  	 11:CASE GVL.mb_Output_Registers[GVL.WATERHARDWARETYPE] OF
		GVL.SWPWTR_TIME:
			//GVL.mb_Output_Registers[GVL.REALTIME_PLC_A2D] :=	0;	//nothing to read with FB circuit, just move motor
			IF GVL.mb_Output_Coils[GVL.REALTIME_ADVANCE] THEN		//move the motor forward
				IF TRUE THEN							//test the FB for limit - can't do this, pass through
					GVL_IO.WaterMotorFwd[FTN1] := TRUE;				// turn on the advance output
					GVL_IO.WaterMotorRvs[FTN1] := FALSE;
					wCycleCount := wCycleCount + 1;
					IF wCycleCount > wMotorTimeOn THEN				//done with timer?
						GVL_IO.WaterMotorFwd[FTN1] := FALSE;		//turn off outputs
						GVL_IO.WaterMotorRvs[FTN1] := FALSE;
						GVL.mb_Output_Coils[GVL.REALTIME_ADVANCE] := FALSE; // reset the advance boolean
						wCycleCount := 0;					//reset the timer counter						
					END_IF
				END_IF
			END_IF
			IF GVL.mb_Output_Coils[GVL.REALTIME_RETARD] THEN
				IF TRUE THEN							//test the FB for limit - can't do this, pass through
					GVL_IO.WaterMotorFwd[FTN1] := FALSE;				// turn on the reverse output
					GVL_IO.WaterMotorRvs[FTN1] := TRUE;
					wCycleCount := wCycleCount + 1;
					IF wCycleCount > wMotorTimeOn THEN				//done with timer?
						GVL_IO.WaterMotorFwd[FTN1] := FALSE;		//turn off outputs
						GVL_IO.WaterMotorRvs[FTN1] := FALSE;
						GVL.mb_Output_Coils[GVL.REALTIME_RETARD] := FALSE; // reset the reverse boolean
						wCycleCount := 0;					//reset the timer counter						
					END_IF
				END_IF
			END_IF
		GVL.SWPWTR_FB:
			GVL.mb_Output_Registers[GVL.REALTIME_PLC_A2D] :=	INT_TO_WORD(GVL_IO.WaterInput[FTN1]);
			IF GVL.mb_Output_Coils[GVL.REALTIME_ADVANCE] THEN		//move the motor forward
				IF GVL_IO.WaterInput[FTN1] < 32000 THEN				//test the FB for limit - assumes 32767 is max of 10 VDC
					GVL_IO.WaterMotorFwd[FTN1] := TRUE;				// turn on the advance output
					GVL_IO.WaterMotorRvs[FTN1] := FALSE;
					wCycleCount := wCycleCount + 1;
					IF wCycleCount > wMotorTimeOn THEN				//done with timer?
						GVL_IO.WaterMotorFwd[FTN1] := FALSE;		//turn off outputs
						GVL_IO.WaterMotorRvs[FTN1] := FALSE;
						GVL.mb_Output_Coils[GVL.REALTIME_ADVANCE] := FALSE; // reset the advance boolean
						wCycleCount := 0;					//reset the timer counter						
						//  curr % sweep   curr ticks - min tick allowed      max sweep %            max ticks allowed      min ticks allowed
						GVL.mb_Output_Registers[GVL.SWEEPTRIMONPRESS + (FTN1 * GVL.WORDRUNTIMEGROUPSIZE)]	:= (INT_TO_WORD(GVL_IO.InkInput[FTN1]) - GVL.w_InkInputIntMin[FTN1]) * 
								(GVL.mb_Output_Registers[GVL.MAXSWEEPTRIM]+1) / (GVL.w_InkInputIntMax[FTN1] - GVL.w_InkInputIntMin[FTN1]);
						//need the onpress setting pointed to the current % sweep of the positioner
					END_IF
				END_IF
			END_IF
			IF GVL.mb_Output_Coils[GVL.REALTIME_RETARD] THEN
				IF GVL_IO.WaterInput[FTN1] > 800 THEN				//test the FB for limit - assumes 32767 is max of 10 VDC
					GVL_IO.WaterMotorFwd[FTN1] := FALSE;				// turn on the reverse output
					GVL_IO.WaterMotorRvs[FTN1] := TRUE;
					wCycleCount := wCycleCount + 1;
					IF wCycleCount > wMotorTimeOn THEN				//done with timer?
						GVL_IO.WaterMotorFwd[FTN1] := FALSE;		//turn off outputs
						GVL_IO.WaterMotorRvs[FTN1] := FALSE;
						GVL.mb_Output_Coils[GVL.REALTIME_RETARD] := FALSE; // reset the reverse boolean
						wCycleCount := 0;					//reset the timer counter						
						//  curr % sweep   curr ticks - min tick allowed      max sweep %            max ticks allowed      min ticks allowed
						GVL.mb_Output_Registers[GVL.SWEEPTRIMONPRESS + (FTN1 * GVL.WORDRUNTIMEGROUPSIZE)]	:= (INT_TO_WORD(GVL_IO.InkInput[FTN1]) - GVL.w_InkInputIntMin[FTN1]) * 
								(GVL.mb_Output_Registers[GVL.MAXSWEEPTRIM]+1) / (GVL.w_InkInputIntMax[FTN1] - GVL.w_InkInputIntMin[FTN1]);
						//need the onpress setting pointed to the current % sweep of the positioner
					END_IF
				END_IF
			END_IF
		GVL.SWPWTR_OUTPUT:
			IF( GVL.b_DINTInput) THEN									//how big should the adv / ret control increment be?
				w_output_incr :=  DINT_TO_INT(GVL.d_DINT10V / 100);
			ELSE
				w_output_incr := (GVL.i_INT10V / 100);
			END_IF
			GVL.mb_Output_Registers[GVL.REALTIME_PLC_A2D] :=	INT_TO_WORD(GVL_IO.WaterSweepOut[FTN1]);
			IF GVL.mb_Output_Coils[GVL.REALTIME_ADVANCE] THEN
				IF GVL_IO.WaterSweepOut[FTN1] < (w_output_incr * 100) THEN
					GVL_IO.WaterSweepOut[FTN1] := GVL_IO.WaterSweepOut[FTN1] + w_output_incr;
				END_IF
				GVL.mb_Output_Coils[GVL.REALTIME_ADVANCE] := FALSE;
			END_IF
			IF GVL.mb_Output_Coils[GVL.REALTIME_RETARD] THEN
				IF GVL_IO.WaterSweepOut[FTN1] > w_output_incr THEN
					GVL_IO.WaterSweepOut[FTN1] := GVL_IO.WaterSweepOut[FTN1] - w_output_incr;
				END_IF
				GVL.mb_Output_Coils[GVL.REALTIME_RETARD] := FALSE;
			END_IF			
		END_CASE
	 12:CASE GVL.mb_Output_Registers[GVL.WATERHARDWARETYPE] OF
		GVL.SWPWTR_TIME:
			//GVL.mb_Output_Registers[GVL.REALTIME_PLC_A2D] :=	0;	//nothing to read with FB circuit, just move motor
			IF GVL.mb_Output_Coils[GVL.REALTIME_ADVANCE] THEN		//move the motor forward
				IF TRUE THEN							//test the FB for limit - can't do this, pass through
					GVL_IO.WaterMotorFwd[FTN2] := TRUE;				// turn on the advance output
					GVL_IO.WaterMotorRvs[FTN2] := FALSE;
					wCycleCount := wCycleCount + 1;
					IF wCycleCount > wMotorTimeOn THEN				//done with timer?
						GVL_IO.WaterMotorFwd[FTN2] := FALSE;		//turn off outputs
						GVL_IO.WaterMotorRvs[FTN2] := FALSE;
						GVL.mb_Output_Coils[GVL.REALTIME_ADVANCE] := FALSE; // reset the advance boolean
						wCycleCount := 0;					//reset the timer counter						
					END_IF
				END_IF
			END_IF
			IF GVL.mb_Output_Coils[GVL.REALTIME_RETARD] THEN
				IF TRUE THEN							//test the FB for limit - can't do this, pass through
					GVL_IO.WaterMotorFwd[FTN2] := FALSE;				// turn on the reverse output
					GVL_IO.WaterMotorRvs[FTN2] := TRUE;
					wCycleCount := wCycleCount + 1;
					IF wCycleCount > wMotorTimeOn THEN				//done with timer?
						GVL_IO.WaterMotorFwd[FTN2] := FALSE;		//turn off outputs
						GVL_IO.WaterMotorRvs[FTN2] := FALSE;
						GVL.mb_Output_Coils[GVL.REALTIME_RETARD] := FALSE; // reset the reverse boolean
						wCycleCount := 0;					//reset the timer counter						
					END_IF
				END_IF
			END_IF
		GVL.SWPWTR_FB:
			GVL.mb_Output_Registers[GVL.REALTIME_PLC_A2D] :=	INT_TO_WORD(GVL_IO.WaterInput[FTN2]);
			IF GVL.mb_Output_Coils[GVL.REALTIME_ADVANCE] THEN		//move the motor forward
				IF GVL_IO.WaterInput[FTN2] < 32000 THEN				//test the FB for limit - assumes 32767 is max of 10 VDC
					GVL_IO.WaterMotorFwd[FTN2] := TRUE;				// turn on the advance output
					GVL_IO.WaterMotorRvs[FTN2] := FALSE;
					wCycleCount := wCycleCount + 1;
					IF wCycleCount > wMotorTimeOn THEN				//done with timer?
						GVL_IO.WaterMotorFwd[FTN2] := FALSE;		//turn off outputs
						GVL_IO.WaterMotorRvs[FTN2] := FALSE;
						GVL.mb_Output_Coils[GVL.REALTIME_ADVANCE] := FALSE; // reset the advance boolean
						wCycleCount := 0;					//reset the timer counter						
						//  curr % sweep   curr ticks - min tick allowed      max sweep %            max ticks allowed      min ticks allowed
						GVL.mb_Output_Registers[GVL.SWEEPTRIMONPRESS + (FTN2 * GVL.WORDRUNTIMEGROUPSIZE)]	:= (INT_TO_WORD(GVL_IO.InkInput[FTN2]) - GVL.w_InkInputIntMin[FTN2]) * 
								(GVL.mb_Output_Registers[GVL.MAXSWEEPTRIM]+1) / (GVL.w_InkInputIntMax[FTN2] - GVL.w_InkInputIntMin[FTN2]);
						//need the onpress setting pointed to the current % sweep of the positioner
					END_IF
				END_IF
			END_IF
			IF GVL.mb_Output_Coils[GVL.REALTIME_RETARD] THEN
				IF GVL_IO.WaterInput[FTN2] > 800 THEN				//test the FB for limit - assumes 32767 is max of 10 VDC
					GVL_IO.WaterMotorFwd[FTN2] := FALSE;				// turn on the reverse output
					GVL_IO.WaterMotorRvs[FTN2] := TRUE;
					wCycleCount := wCycleCount + 1;
					IF wCycleCount > wMotorTimeOn THEN				//done with timer?
						GVL_IO.WaterMotorFwd[FTN2] := FALSE;		//turn off outputs
						GVL_IO.WaterMotorRvs[FTN2] := FALSE;
						GVL.mb_Output_Coils[GVL.REALTIME_RETARD] := FALSE; // reset the reverse boolean
						wCycleCount := 0;					//reset the timer counter						
						//  curr % sweep   curr ticks - min tick allowed      max sweep %            max ticks allowed      min ticks allowed
						GVL.mb_Output_Registers[GVL.SWEEPTRIMONPRESS + (FTN2 * GVL.WORDRUNTIMEGROUPSIZE)]	:= (INT_TO_WORD(GVL_IO.InkInput[FTN2]) - GVL.w_InkInputIntMin[FTN2]) * 
								(GVL.mb_Output_Registers[GVL.MAXSWEEPTRIM]+1) / (GVL.w_InkInputIntMax[FTN2] - GVL.w_InkInputIntMin[FTN2]);
						//need the onpress setting pointed to the current % sweep of the positioner
					END_IF
				END_IF
			END_IF
		GVL.SWPWTR_OUTPUT:
			IF( GVL.b_DINTInput) THEN									//how big should the adv / ret control increment be?
				w_output_incr :=  DINT_TO_INT(GVL.d_DINT10V / 100);
			ELSE
				w_output_incr := (GVL.i_INT10V / 100);
			END_IF
			GVL.mb_Output_Registers[GVL.REALTIME_PLC_A2D] :=	INT_TO_WORD(GVL_IO.WaterSweepOut[FTN2]);
			IF GVL.mb_Output_Coils[GVL.REALTIME_ADVANCE] THEN
				IF GVL_IO.WaterSweepOut[FTN2] < (w_output_incr * 100) THEN
					GVL_IO.WaterSweepOut[FTN2] := GVL_IO.WaterSweepOut[FTN2] + w_output_incr;
				END_IF
				GVL.mb_Output_Coils[GVL.REALTIME_ADVANCE] := FALSE;
			END_IF
			IF GVL.mb_Output_Coils[GVL.REALTIME_RETARD] THEN
				IF GVL_IO.WaterSweepOut[FTN2] > w_output_incr THEN
					GVL_IO.WaterSweepOut[FTN2] := GVL_IO.WaterSweepOut[FTN2] - w_output_incr;
				END_IF
				GVL.mb_Output_Coils[GVL.REALTIME_RETARD] := FALSE;
			END_IF			
		END_CASE
	 13:CASE GVL.mb_Output_Registers[GVL.WATERHARDWARETYPE] OF
		GVL.SWPWTR_TIME:
			//GVL.mb_Output_Registers[GVL.REALTIME_PLC_A2D] :=	0;	//nothing to read with FB circuit, just move motor
			IF GVL.mb_Output_Coils[GVL.REALTIME_ADVANCE] THEN		//move the motor forward
				IF TRUE THEN							//test the FB for limit - can't do this, pass through
					GVL_IO.WaterMotorFwd[FTN3] := TRUE;				// turn on the advance output
					GVL_IO.WaterMotorRvs[FTN3] := FALSE;
					wCycleCount := wCycleCount + 1;
					IF wCycleCount > wMotorTimeOn THEN				//done with timer?
						GVL_IO.WaterMotorFwd[FTN3] := FALSE;		//turn off outputs
						GVL_IO.WaterMotorRvs[FTN3] := FALSE;
						GVL.mb_Output_Coils[GVL.REALTIME_ADVANCE] := FALSE; // reset the advance boolean
						wCycleCount := 0;					//reset the timer counter						
					END_IF
				END_IF
			END_IF
			IF GVL.mb_Output_Coils[GVL.REALTIME_RETARD] THEN
				IF TRUE THEN							//test the FB for limit - can't do this, pass through
					GVL_IO.WaterMotorFwd[FTN3] := FALSE;				// turn on the reverse output
					GVL_IO.WaterMotorRvs[FTN3] := TRUE;
					wCycleCount := wCycleCount + 1;
					IF wCycleCount > wMotorTimeOn THEN				//done with timer?
						GVL_IO.WaterMotorFwd[FTN3] := FALSE;		//turn off outputs
						GVL_IO.WaterMotorRvs[FTN3] := FALSE;
						GVL.mb_Output_Coils[GVL.REALTIME_RETARD] := FALSE; // reset the reverse boolean
						wCycleCount := 0;					//reset the timer counter						
					END_IF
				END_IF
			END_IF
		GVL.SWPWTR_FB:
			GVL.mb_Output_Registers[GVL.REALTIME_PLC_A2D] :=	INT_TO_WORD(GVL_IO.WaterInput[FTN3]);
			IF GVL.mb_Output_Coils[GVL.REALTIME_ADVANCE] THEN		//move the motor forward
				IF GVL_IO.WaterInput[FTN3] < 32000 THEN				//test the FB for limit - assumes 32767 is max of 10 VDC
					GVL_IO.WaterMotorFwd[FTN3] := TRUE;				// turn on the advance output
					GVL_IO.WaterMotorRvs[FTN3] := FALSE;
					wCycleCount := wCycleCount + 1;
					IF wCycleCount > wMotorTimeOn THEN				//done with timer?
						GVL_IO.WaterMotorFwd[FTN3] := FALSE;		//turn off outputs
						GVL_IO.WaterMotorRvs[FTN3] := FALSE;
						GVL.mb_Output_Coils[GVL.REALTIME_ADVANCE] := FALSE; // reset the advance boolean
						wCycleCount := 0;					//reset the timer counter						
						//  curr % sweep   curr ticks - min tick allowed      max sweep %            max ticks allowed      min ticks allowed
						GVL.mb_Output_Registers[GVL.SWEEPTRIMONPRESS + (FTN3 * GVL.WORDRUNTIMEGROUPSIZE)]	:= (INT_TO_WORD(GVL_IO.InkInput[FTN3]) - GVL.w_InkInputIntMin[FTN3]) * 
								(GVL.mb_Output_Registers[GVL.MAXSWEEPTRIM]+1) / (GVL.w_InkInputIntMax[FTN3] - GVL.w_InkInputIntMin[FTN3]);
						//need the onpress setting pointed to the current % sweep of the positioner
					END_IF
				END_IF
			END_IF
			IF GVL.mb_Output_Coils[GVL.REALTIME_RETARD] THEN
				IF GVL_IO.WaterInput[FTN3] > 800 THEN				//test the FB for limit - assumes 32767 is max of 10 VDC
					GVL_IO.WaterMotorFwd[FTN3] := FALSE;				// turn on the reverse output
					GVL_IO.WaterMotorRvs[FTN3] := TRUE;
					wCycleCount := wCycleCount + 1;
					IF wCycleCount > wMotorTimeOn THEN				//done with timer?
						GVL_IO.WaterMotorFwd[FTN3] := FALSE;		//turn off outputs
						GVL_IO.WaterMotorRvs[FTN3] := FALSE;
						GVL.mb_Output_Coils[GVL.REALTIME_RETARD] := FALSE; // reset the reverse boolean
						wCycleCount := 0;					//reset the timer counter						
						//  curr % sweep   curr ticks - min tick allowed      max sweep %            max ticks allowed      min ticks allowed
						GVL.mb_Output_Registers[GVL.SWEEPTRIMONPRESS + (FTN3 * GVL.WORDRUNTIMEGROUPSIZE)]	:= (INT_TO_WORD(GVL_IO.InkInput[FTN3]) - GVL.w_InkInputIntMin[FTN3]) * 
								(GVL.mb_Output_Registers[GVL.MAXSWEEPTRIM]+1) / (GVL.w_InkInputIntMax[FTN3] - GVL.w_InkInputIntMin[FTN3]);
						//need the onpress setting pointed to the current % sweep of the positioner
					END_IF
				END_IF
			END_IF
		GVL.SWPWTR_OUTPUT:
			IF( GVL.b_DINTInput) THEN									//how big should the adv / ret control increment be?
				w_output_incr :=  DINT_TO_INT(GVL.d_DINT10V / 100);
			ELSE
				w_output_incr := (GVL.i_INT10V / 100);
			END_IF
			GVL.mb_Output_Registers[GVL.REALTIME_PLC_A2D] :=	INT_TO_WORD(GVL_IO.WaterSweepOut[FTN3]);
			IF GVL.mb_Output_Coils[GVL.REALTIME_ADVANCE] THEN
				IF GVL_IO.WaterSweepOut[FTN3] < (w_output_incr * 100) THEN
					GVL_IO.WaterSweepOut[FTN3] := GVL_IO.WaterSweepOut[FTN3] + w_output_incr;
				END_IF
				GVL.mb_Output_Coils[GVL.REALTIME_ADVANCE] := FALSE;
			END_IF
			IF GVL.mb_Output_Coils[GVL.REALTIME_RETARD] THEN
				IF GVL_IO.WaterSweepOut[FTN3] > w_output_incr THEN
					GVL_IO.WaterSweepOut[FTN3] := GVL_IO.WaterSweepOut[FTN3] - w_output_incr;
				END_IF
				GVL.mb_Output_Coils[GVL.REALTIME_RETARD] := FALSE;
			END_IF			
		END_CASE
	 14:CASE GVL.mb_Output_Registers[GVL.WATERHARDWARETYPE] OF
		GVL.SWPWTR_TIME:
			//GVL.mb_Output_Registers[GVL.REALTIME_PLC_A2D] :=	0;	//nothing to read with FB circuit, just move motor
			IF GVL.mb_Output_Coils[GVL.REALTIME_ADVANCE] THEN		//move the motor forward
				IF TRUE THEN							//test the FB for limit - can't do this, pass through
					GVL_IO.WaterMotorFwd[FTN4] := TRUE;				// turn on the advance output
					GVL_IO.WaterMotorRvs[FTN4] := FALSE;
					wCycleCount := wCycleCount + 1;
					IF wCycleCount > wMotorTimeOn THEN				//done with timer?
						GVL_IO.WaterMotorFwd[FTN4] := FALSE;		//turn off outputs
						GVL_IO.WaterMotorRvs[FTN4] := FALSE;
						GVL.mb_Output_Coils[GVL.REALTIME_ADVANCE] := FALSE; // reset the advance boolean
						wCycleCount := 0;					//reset the timer counter						
					END_IF
				END_IF
			END_IF
			IF GVL.mb_Output_Coils[GVL.REALTIME_RETARD] THEN
				IF TRUE THEN							//test the FB for limit - can't do this, pass through
					GVL_IO.WaterMotorFwd[FTN4] := FALSE;				// turn on the reverse output
					GVL_IO.WaterMotorRvs[FTN4] := TRUE;
					wCycleCount := wCycleCount + 1;
					IF wCycleCount > wMotorTimeOn THEN				//done with timer?
						GVL_IO.WaterMotorFwd[FTN4] := FALSE;		//turn off outputs
						GVL_IO.WaterMotorRvs[FTN4] := FALSE;
						GVL.mb_Output_Coils[GVL.REALTIME_RETARD] := FALSE; // reset the reverse boolean
						wCycleCount := 0;					//reset the timer counter						
					END_IF
				END_IF
			END_IF
		GVL.SWPWTR_FB:
			GVL.mb_Output_Registers[GVL.REALTIME_PLC_A2D] :=	INT_TO_WORD(GVL_IO.WaterInput[FTN4]);
			IF GVL.mb_Output_Coils[GVL.REALTIME_ADVANCE] THEN		//move the motor forward
				IF GVL_IO.WaterInput[FTN4] < 32000 THEN				//test the FB for limit - assumes 32767 is max of 10 VDC
					GVL_IO.WaterMotorFwd[FTN4] := TRUE;				// turn on the advance output
					GVL_IO.WaterMotorRvs[FTN4] := FALSE;
					wCycleCount := wCycleCount + 1;
					IF wCycleCount > wMotorTimeOn THEN				//done with timer?
						GVL_IO.WaterMotorFwd[FTN4] := FALSE;		//turn off outputs
						GVL_IO.WaterMotorRvs[FTN4] := FALSE;
						GVL.mb_Output_Coils[GVL.REALTIME_ADVANCE] := FALSE; // reset the advance boolean
						wCycleCount := 0;					//reset the timer counter						
						//  curr % sweep   curr ticks - min tick allowed      max sweep %            max ticks allowed      min ticks allowed
						GVL.mb_Output_Registers[GVL.SWEEPTRIMONPRESS + (FTN4 * GVL.WORDRUNTIMEGROUPSIZE)]	:= (INT_TO_WORD(GVL_IO.InkInput[FTN4]) - GVL.w_InkInputIntMin[FTN4]) * 
								(GVL.mb_Output_Registers[GVL.MAXSWEEPTRIM]+1) / (GVL.w_InkInputIntMax[FTN4] - GVL.w_InkInputIntMin[FTN4]);
						//need the onpress setting pointed to the current % sweep of the positioner
					END_IF
				END_IF
			END_IF
			IF GVL.mb_Output_Coils[GVL.REALTIME_RETARD] THEN
				IF GVL_IO.WaterInput[FTN4] > 800 THEN				//test the FB for limit - assumes 32767 is max of 10 VDC
					GVL_IO.WaterMotorFwd[FTN4] := FALSE;				// turn on the reverse output
					GVL_IO.WaterMotorRvs[FTN4] := TRUE;
					wCycleCount := wCycleCount + 1;
					IF wCycleCount > wMotorTimeOn THEN				//done with timer?
						GVL_IO.WaterMotorFwd[FTN4] := FALSE;		//turn off outputs
						GVL_IO.WaterMotorRvs[FTN4] := FALSE;
						GVL.mb_Output_Coils[GVL.REALTIME_RETARD] := FALSE; // reset the reverse boolean
						wCycleCount := 0;					//reset the timer counter						
						//  curr % sweep   curr ticks - min tick allowed      max sweep %            max ticks allowed      min ticks allowed
						GVL.mb_Output_Registers[GVL.SWEEPTRIMONPRESS + (FTN4 * GVL.WORDRUNTIMEGROUPSIZE)]	:= (INT_TO_WORD(GVL_IO.InkInput[FTN4]) - GVL.w_InkInputIntMin[FTN4]) * 
								(GVL.mb_Output_Registers[GVL.MAXSWEEPTRIM]+1) / (GVL.w_InkInputIntMax[FTN4] - GVL.w_InkInputIntMin[FTN4]);
						//need the onpress setting pointed to the current % sweep of the positioner
					END_IF
				END_IF
			END_IF
		GVL.SWPWTR_OUTPUT:
			IF( GVL.b_DINTInput) THEN									//how big should the adv / ret control increment be?
				w_output_incr :=  DINT_TO_INT(GVL.d_DINT10V / 100);
			ELSE
				w_output_incr := (GVL.i_INT10V / 100);
			END_IF
			GVL.mb_Output_Registers[GVL.REALTIME_PLC_A2D] :=	INT_TO_WORD(GVL_IO.WaterSweepOut[FTN4]);
			IF GVL.mb_Output_Coils[GVL.REALTIME_ADVANCE] THEN
				IF GVL_IO.WaterSweepOut[FTN4] < (w_output_incr * 100) THEN
					GVL_IO.WaterSweepOut[FTN4] := GVL_IO.WaterSweepOut[FTN4] + w_output_incr;
				END_IF
				GVL.mb_Output_Coils[GVL.REALTIME_ADVANCE] := FALSE;
			END_IF
			IF GVL.mb_Output_Coils[GVL.REALTIME_RETARD] THEN
				IF GVL_IO.WaterSweepOut[FTN4] > w_output_incr THEN
					GVL_IO.WaterSweepOut[FTN4] := GVL_IO.WaterSweepOut[FTN4] - w_output_incr;
				END_IF
				GVL.mb_Output_Coils[GVL.REALTIME_RETARD] := FALSE;
			END_IF			
		END_CASE
	 15:CASE GVL.mb_Output_Registers[GVL.WATERHARDWARETYPE] OF
		GVL.SWPWTR_TIME:
			//GVL.mb_Output_Registers[GVL.REALTIME_PLC_A2D] :=	0;	//nothing to read with FB circuit, just move motor
			IF GVL.mb_Output_Coils[GVL.REALTIME_ADVANCE] THEN		//move the motor forward
				IF TRUE THEN							//test the FB for limit - can't do this, pass through
					GVL_IO.WaterMotorFwd[FTN5] := TRUE;				// turn on the advance output
					GVL_IO.WaterMotorRvs[FTN5] := FALSE;
					wCycleCount := wCycleCount + 1;
					IF wCycleCount > wMotorTimeOn THEN				//done with timer?
						GVL_IO.WaterMotorFwd[FTN5] := FALSE;		//turn off outputs
						GVL_IO.WaterMotorRvs[FTN5] := FALSE;
						GVL.mb_Output_Coils[GVL.REALTIME_ADVANCE] := FALSE; // reset the advance boolean
						wCycleCount := 0;					//reset the timer counter						
					END_IF
				END_IF
			END_IF
			IF GVL.mb_Output_Coils[GVL.REALTIME_RETARD] THEN
				IF TRUE THEN							//test the FB for limit - can't do this, pass through
					GVL_IO.WaterMotorFwd[FTN5] := FALSE;				// turn on the reverse output
					GVL_IO.WaterMotorRvs[FTN5] := TRUE;
					wCycleCount := wCycleCount + 1;
					IF wCycleCount > wMotorTimeOn THEN				//done with timer?
						GVL_IO.WaterMotorFwd[FTN5] := FALSE;		//turn off outputs
						GVL_IO.WaterMotorRvs[FTN5] := FALSE;
						GVL.mb_Output_Coils[GVL.REALTIME_RETARD] := FALSE; // reset the reverse boolean
						wCycleCount := 0;					//reset the timer counter						
					END_IF
				END_IF
			END_IF
		GVL.SWPWTR_FB:
			GVL.mb_Output_Registers[GVL.REALTIME_PLC_A2D] :=	INT_TO_WORD(GVL_IO.WaterInput[FTN5]);
			IF GVL.mb_Output_Coils[GVL.REALTIME_ADVANCE] THEN		//move the motor forward
				IF GVL_IO.WaterInput[FTN5] < 32000 THEN				//test the FB for limit - assumes 32767 is max of 10 VDC
					GVL_IO.WaterMotorFwd[FTN5] := TRUE;				// turn on the advance output
					GVL_IO.WaterMotorRvs[FTN5] := FALSE;
					wCycleCount := wCycleCount + 1;
					IF wCycleCount > wMotorTimeOn THEN				//done with timer?
						GVL_IO.WaterMotorFwd[FTN5] := FALSE;		//turn off outputs
						GVL_IO.WaterMotorRvs[FTN5] := FALSE;
						GVL.mb_Output_Coils[GVL.REALTIME_ADVANCE] := FALSE; // reset the advance boolean
						wCycleCount := 0;					//reset the timer counter						
						//  curr % sweep   curr ticks - min tick allowed      max sweep %            max ticks allowed      min ticks allowed
						GVL.mb_Output_Registers[GVL.SWEEPTRIMONPRESS + (FTN5 * GVL.WORDRUNTIMEGROUPSIZE)]	:= (INT_TO_WORD(GVL_IO.InkInput[FTN5]) - GVL.w_InkInputIntMin[FTN5]) * 
								(GVL.mb_Output_Registers[GVL.MAXSWEEPTRIM]+1) / (GVL.w_InkInputIntMax[FTN5] - GVL.w_InkInputIntMin[FTN5]);
						//need the onpress setting pointed to the current % sweep of the positioner
					END_IF
				END_IF
			END_IF
			IF GVL.mb_Output_Coils[GVL.REALTIME_RETARD] THEN
				IF GVL_IO.WaterInput[FTN5] > 800 THEN				//test the FB for limit - assumes 32767 is max of 10 VDC
					GVL_IO.WaterMotorFwd[FTN5] := FALSE;				// turn on the reverse output
					GVL_IO.WaterMotorRvs[FTN5] := TRUE;
					wCycleCount := wCycleCount + 1;
					IF wCycleCount > wMotorTimeOn THEN				//done with timer?
						GVL_IO.WaterMotorFwd[FTN5] := FALSE;		//turn off outputs
						GVL_IO.WaterMotorRvs[FTN5] := FALSE;
						GVL.mb_Output_Coils[GVL.REALTIME_RETARD] := FALSE; // reset the reverse boolean
						wCycleCount := 0;					//reset the timer counter						
						//  curr % sweep   curr ticks - min tick allowed      max sweep %            max ticks allowed      min ticks allowed
						GVL.mb_Output_Registers[GVL.SWEEPTRIMONPRESS + (FTN5 * GVL.WORDRUNTIMEGROUPSIZE)]	:= (INT_TO_WORD(GVL_IO.InkInput[FTN5]) - GVL.w_InkInputIntMin[FTN5]) * 
								(GVL.mb_Output_Registers[GVL.MAXSWEEPTRIM]+1) / (GVL.w_InkInputIntMax[FTN5] - GVL.w_InkInputIntMin[FTN5]);
						//need the onpress setting pointed to the current % sweep of the positioner
					END_IF
				END_IF
			END_IF
		GVL.SWPWTR_OUTPUT:
			IF( GVL.b_DINTInput) THEN									//how big should the adv / ret control increment be?
				w_output_incr :=  DINT_TO_INT(GVL.d_DINT10V / 100);
			ELSE
				w_output_incr := (GVL.i_INT10V / 100);
			END_IF
			GVL.mb_Output_Registers[GVL.REALTIME_PLC_A2D] :=	INT_TO_WORD(GVL_IO.WaterSweepOut[FTN5]);
			IF GVL.mb_Output_Coils[GVL.REALTIME_ADVANCE] THEN
				IF GVL_IO.WaterSweepOut[FTN5] < (w_output_incr * 100) THEN
					GVL_IO.WaterSweepOut[FTN5] := GVL_IO.WaterSweepOut[FTN5] + w_output_incr;
				END_IF
				GVL.mb_Output_Coils[GVL.REALTIME_ADVANCE] := FALSE;
			END_IF
			IF GVL.mb_Output_Coils[GVL.REALTIME_RETARD] THEN
				IF GVL_IO.WaterSweepOut[FTN5] > w_output_incr THEN
					GVL_IO.WaterSweepOut[FTN5] := GVL_IO.WaterSweepOut[FTN5] - w_output_incr;
				END_IF
				GVL.mb_Output_Coils[GVL.REALTIME_RETARD] := FALSE;
			END_IF			
		END_CASE
	 16:CASE GVL.mb_Output_Registers[GVL.WATERHARDWARETYPE] OF
		GVL.SWPWTR_TIME:
			//GVL.mb_Output_Registers[GVL.REALTIME_PLC_A2D] :=	0;	//nothing to read with FB circuit, just move motor
			IF GVL.mb_Output_Coils[GVL.REALTIME_ADVANCE] THEN		//move the motor forward
				IF TRUE THEN							//test the FB for limit - can't do this, pass through
					GVL_IO.WaterMotorFwd[FTN6] := TRUE;				// turn on the advance output
					GVL_IO.WaterMotorRvs[FTN6] := FALSE;
					wCycleCount := wCycleCount + 1;
					IF wCycleCount > wMotorTimeOn THEN				//done with timer?
						GVL_IO.WaterMotorFwd[FTN6] := FALSE;		//turn off outputs
						GVL_IO.WaterMotorRvs[FTN6] := FALSE;
						GVL.mb_Output_Coils[GVL.REALTIME_ADVANCE] := FALSE; // reset the advance boolean
						wCycleCount := 0;					//reset the timer counter						
					END_IF
				END_IF
			END_IF
			IF GVL.mb_Output_Coils[GVL.REALTIME_RETARD] THEN
				IF TRUE THEN							//test the FB for limit - can't do this, pass through
					GVL_IO.WaterMotorFwd[FTN6] := FALSE;				// turn on the reverse output
					GVL_IO.WaterMotorRvs[FTN6] := TRUE;
					wCycleCount := wCycleCount + 1;
					IF wCycleCount > wMotorTimeOn THEN				//done with timer?
						GVL_IO.WaterMotorFwd[FTN6] := FALSE;		//turn off outputs
						GVL_IO.WaterMotorRvs[FTN6] := FALSE;
						GVL.mb_Output_Coils[GVL.REALTIME_RETARD] := FALSE; // reset the reverse boolean
						wCycleCount := 0;					//reset the timer counter						
					END_IF
				END_IF
			END_IF
		GVL.SWPWTR_FB:
			GVL.mb_Output_Registers[GVL.REALTIME_PLC_A2D] :=	INT_TO_WORD(GVL_IO.WaterInput[FTN6]);
			IF GVL.mb_Output_Coils[GVL.REALTIME_ADVANCE] THEN		//move the motor forward
				IF GVL_IO.WaterInput[FTN6] < 32000 THEN				//test the FB for limit - assumes 32767 is max of 10 VDC
					GVL_IO.WaterMotorFwd[FTN6] := TRUE;				// turn on the advance output
					GVL_IO.WaterMotorRvs[FTN6] := FALSE;
					wCycleCount := wCycleCount + 1;
					IF wCycleCount > wMotorTimeOn THEN				//done with timer?
						GVL_IO.WaterMotorFwd[FTN6] := FALSE;		//turn off outputs
						GVL_IO.WaterMotorRvs[FTN6] := FALSE;
						GVL.mb_Output_Coils[GVL.REALTIME_ADVANCE] := FALSE; // reset the advance boolean
						wCycleCount := 0;					//reset the timer counter						
						//  curr % sweep   curr ticks - min tick allowed      max sweep %            max ticks allowed      min ticks allowed
						GVL.mb_Output_Registers[GVL.SWEEPTRIMONPRESS + (FTN6 * GVL.WORDRUNTIMEGROUPSIZE)]	:= (INT_TO_WORD(GVL_IO.InkInput[FTN6]) - GVL.w_InkInputIntMin[FTN6]) * 
								(GVL.mb_Output_Registers[GVL.MAXSWEEPTRIM]+1) / (GVL.w_InkInputIntMax[FTN6] - GVL.w_InkInputIntMin[FTN6]);
						//need the onpress setting pointed to the current % sweep of the positioner
					END_IF
				END_IF
			END_IF
			IF GVL.mb_Output_Coils[GVL.REALTIME_RETARD] THEN
				IF GVL_IO.WaterInput[FTN6] > 800 THEN				//test the FB for limit - assumes 32767 is max of 10 VDC
					GVL_IO.WaterMotorFwd[FTN6] := FALSE;				// turn on the reverse output
					GVL_IO.WaterMotorRvs[FTN6] := TRUE;
					wCycleCount := wCycleCount + 1;
					IF wCycleCount > wMotorTimeOn THEN				//done with timer?
						GVL_IO.WaterMotorFwd[FTN6] := FALSE;		//turn off outputs
						GVL_IO.WaterMotorRvs[FTN6] := FALSE;
						GVL.mb_Output_Coils[GVL.REALTIME_RETARD] := FALSE; // reset the reverse boolean
						wCycleCount := 0;					//reset the timer counter						
						//  curr % sweep   curr ticks - min tick allowed      max sweep %            max ticks allowed      min ticks allowed
						GVL.mb_Output_Registers[GVL.SWEEPTRIMONPRESS + (FTN6 * GVL.WORDRUNTIMEGROUPSIZE)]	:= (INT_TO_WORD(GVL_IO.InkInput[FTN6]) - GVL.w_InkInputIntMin[FTN6]) * 
								(GVL.mb_Output_Registers[GVL.MAXSWEEPTRIM]+1) / (GVL.w_InkInputIntMax[FTN6] - GVL.w_InkInputIntMin[FTN6]);
						//need the onpress setting pointed to the current % sweep of the positioner
					END_IF
				END_IF
			END_IF
		GVL.SWPWTR_OUTPUT:
			IF( GVL.b_DINTInput) THEN									//how big should the adv / ret control increment be?
				w_output_incr :=  DINT_TO_INT(GVL.d_DINT10V / 100);
			ELSE
				w_output_incr := (GVL.i_INT10V / 100);
			END_IF
			GVL.mb_Output_Registers[GVL.REALTIME_PLC_A2D] :=	INT_TO_WORD(GVL_IO.WaterSweepOut[FTN6]);
			IF GVL.mb_Output_Coils[GVL.REALTIME_ADVANCE] THEN
				IF GVL_IO.WaterSweepOut[FTN6] < (w_output_incr * 100) THEN
					GVL_IO.WaterSweepOut[FTN6] := GVL_IO.WaterSweepOut[FTN6] + w_output_incr;
				END_IF
				GVL.mb_Output_Coils[GVL.REALTIME_ADVANCE] := FALSE;
			END_IF
			IF GVL.mb_Output_Coils[GVL.REALTIME_RETARD] THEN
				IF GVL_IO.WaterSweepOut[FTN6] > w_output_incr THEN
					GVL_IO.WaterSweepOut[FTN6] := GVL_IO.WaterSweepOut[FTN6] - w_output_incr;
				END_IF
				GVL.mb_Output_Coils[GVL.REALTIME_RETARD] := FALSE;
			END_IF			
		END_CASE
	 17:CASE GVL.mb_Output_Registers[GVL.WATERHARDWARETYPE] OF
		GVL.SWPWTR_TIME:
			//GVL.mb_Output_Registers[GVL.REALTIME_PLC_A2D] :=	0;	//nothing to read with FB circuit, just move motor
			IF GVL.mb_Output_Coils[GVL.REALTIME_ADVANCE] THEN		//move the motor forward
				IF TRUE THEN							//test the FB for limit - can't do this, pass through
					GVL_IO.WaterMotorFwd[FTN7] := TRUE;				// turn on the advance output
					GVL_IO.WaterMotorRvs[FTN7] := FALSE;
					wCycleCount := wCycleCount + 1;
					IF wCycleCount > wMotorTimeOn THEN				//done with timer?
						GVL_IO.WaterMotorFwd[FTN7] := FALSE;		//turn off outputs
						GVL_IO.WaterMotorRvs[FTN7] := FALSE;
						GVL.mb_Output_Coils[GVL.REALTIME_ADVANCE] := FALSE; // reset the advance boolean
						wCycleCount := 0;					//reset the timer counter						
					END_IF
				END_IF
			END_IF
			IF GVL.mb_Output_Coils[GVL.REALTIME_RETARD] THEN
				IF TRUE THEN							//test the FB for limit - can't do this, pass through
					GVL_IO.WaterMotorFwd[FTN7] := FALSE;				// turn on the reverse output
					GVL_IO.WaterMotorRvs[FTN7] := TRUE;
					wCycleCount := wCycleCount + 1;
					IF wCycleCount > wMotorTimeOn THEN				//done with timer?
						GVL_IO.WaterMotorFwd[FTN7] := FALSE;		//turn off outputs
						GVL_IO.WaterMotorRvs[FTN7] := FALSE;
						GVL.mb_Output_Coils[GVL.REALTIME_RETARD] := FALSE; // reset the reverse boolean
						wCycleCount := 0;					//reset the timer counter						
					END_IF
				END_IF
			END_IF
		GVL.SWPWTR_FB:
			GVL.mb_Output_Registers[GVL.REALTIME_PLC_A2D] :=	INT_TO_WORD(GVL_IO.WaterInput[FTN7]);
			IF GVL.mb_Output_Coils[GVL.REALTIME_ADVANCE] THEN		//move the motor forward
				IF GVL_IO.WaterInput[FTN7] < 32000 THEN				//test the FB for limit - assumes 32767 is max of 10 VDC
					GVL_IO.WaterMotorFwd[FTN7] := TRUE;				// turn on the advance output
					GVL_IO.WaterMotorRvs[FTN7] := FALSE;
					wCycleCount := wCycleCount + 1;
					IF wCycleCount > wMotorTimeOn THEN				//done with timer?
						GVL_IO.WaterMotorFwd[FTN7] := FALSE;		//turn off outputs
						GVL_IO.WaterMotorRvs[FTN7] := FALSE;
						GVL.mb_Output_Coils[GVL.REALTIME_ADVANCE] := FALSE; // reset the advance boolean
						wCycleCount := 0;					//reset the timer counter						
						//  curr % sweep   curr ticks - min tick allowed      max sweep %            max ticks allowed      min ticks allowed
						GVL.mb_Output_Registers[GVL.SWEEPTRIMONPRESS + Index_offset + (FTN7 * GVL.WORDRUNTIMEGROUPSIZE)]	:= (INT_TO_WORD(GVL_IO.InkInput[FTN7]) - GVL.w_InkInputIntMin[FTN7]) * 
								(GVL.mb_Output_Registers[GVL.MAXSWEEPTRIM]+1) / (GVL.w_InkInputIntMax[FTN7] - GVL.w_InkInputIntMin[FTN7]);
						//need the onpress setting pointed to the current % sweep of the positioner
					END_IF
				END_IF
			END_IF
			IF GVL.mb_Output_Coils[GVL.REALTIME_RETARD] THEN
				IF GVL_IO.WaterInput[FTN7] > 800 THEN				//test the FB for limit - assumes 32767 is max of 10 VDC
					GVL_IO.WaterMotorFwd[FTN7] := FALSE;				// turn on the reverse output
					GVL_IO.WaterMotorRvs[FTN7] := TRUE;
					wCycleCount := wCycleCount + 1;
					IF wCycleCount > wMotorTimeOn THEN				//done with timer?
						GVL_IO.WaterMotorFwd[FTN7] := FALSE;		//turn off outputs
						GVL_IO.WaterMotorRvs[FTN7] := FALSE;
						GVL.mb_Output_Coils[GVL.REALTIME_RETARD] := FALSE; // reset the reverse boolean
						wCycleCount := 0;					//reset the timer counter						
						//  curr % sweep   curr ticks - min tick allowed      max sweep %            max ticks allowed      min ticks allowed
						GVL.mb_Output_Registers[GVL.SWEEPTRIMONPRESS + Index_offset + (FTN7 * GVL.WORDRUNTIMEGROUPSIZE)]	:= (INT_TO_WORD(GVL_IO.InkInput[FTN7]) - GVL.w_InkInputIntMin[FTN7]) * 
								(GVL.mb_Output_Registers[GVL.MAXSWEEPTRIM]+1) / (GVL.w_InkInputIntMax[FTN7] - GVL.w_InkInputIntMin[FTN7]);
						//need the onpress setting pointed to the current % sweep of the positioner
					END_IF
				END_IF
			END_IF
		GVL.SWPWTR_OUTPUT:
			IF( GVL.b_DINTInput) THEN									//how big should the adv / ret control increment be?
				w_output_incr :=  DINT_TO_INT(GVL.d_DINT10V / 100);
			ELSE
				w_output_incr := (GVL.i_INT10V / 100);
			END_IF
			GVL.mb_Output_Registers[GVL.REALTIME_PLC_A2D] :=	INT_TO_WORD(GVL_IO.WaterSweepOut[FTN7]);
			IF GVL.mb_Output_Coils[GVL.REALTIME_ADVANCE] THEN
				IF GVL_IO.WaterSweepOut[FTN7] < (w_output_incr * 100) THEN
					GVL_IO.WaterSweepOut[FTN7] := GVL_IO.WaterSweepOut[FTN7] + w_output_incr;
				END_IF
				GVL.mb_Output_Coils[GVL.REALTIME_ADVANCE] := FALSE;
			END_IF
			IF GVL.mb_Output_Coils[GVL.REALTIME_RETARD] THEN
				IF GVL_IO.WaterSweepOut[FTN7] > w_output_incr THEN
					GVL_IO.WaterSweepOut[FTN7] := GVL_IO.WaterSweepOut[FTN7] - w_output_incr;
				END_IF
				GVL.mb_Output_Coils[GVL.REALTIME_RETARD] := FALSE;
			END_IF			
		END_CASE
	 18:CASE GVL.mb_Output_Registers[GVL.WATERHARDWARETYPE] OF
		GVL.SWPWTR_TIME:
			//GVL.mb_Output_Registers[GVL.REALTIME_PLC_A2D] :=	0;	//nothing to read with FB circuit, just move motor
			IF GVL.mb_Output_Coils[GVL.REALTIME_ADVANCE] THEN		//move the motor forward
				IF TRUE THEN							//test the FB for limit - can't do this, pass through
					GVL_IO.WaterMotorFwd[FTN8] := TRUE;				// turn on the advance output
					GVL_IO.WaterMotorRvs[FTN8] := FALSE;
					wCycleCount := wCycleCount + 1;
					IF wCycleCount > wMotorTimeOn THEN				//done with timer?
						GVL_IO.WaterMotorFwd[FTN8] := FALSE;		//turn off outputs
						GVL_IO.WaterMotorRvs[FTN8] := FALSE;
						GVL.mb_Output_Coils[GVL.REALTIME_ADVANCE] := FALSE; // reset the advance boolean
						wCycleCount := 0;					//reset the timer counter						
					END_IF
				END_IF
			END_IF
			IF GVL.mb_Output_Coils[GVL.REALTIME_RETARD] THEN
				IF TRUE THEN							//test the FB for limit - can't do this, pass through
					GVL_IO.WaterMotorFwd[FTN8] := FALSE;				// turn on the reverse output
					GVL_IO.WaterMotorRvs[FTN8] := TRUE;
					wCycleCount := wCycleCount + 1;
					IF wCycleCount > wMotorTimeOn THEN				//done with timer?
						GVL_IO.WaterMotorFwd[FTN8] := FALSE;		//turn off outputs
						GVL_IO.WaterMotorRvs[FTN8] := FALSE;
						GVL.mb_Output_Coils[GVL.REALTIME_RETARD] := FALSE; // reset the reverse boolean
						wCycleCount := 0;					//reset the timer counter						
					END_IF
				END_IF
			END_IF
		GVL.SWPWTR_FB:
			GVL.mb_Output_Registers[GVL.REALTIME_PLC_A2D] :=	INT_TO_WORD(GVL_IO.WaterInput[FTN8]);
			IF GVL.mb_Output_Coils[GVL.REALTIME_ADVANCE] THEN		//move the motor forward
				IF GVL_IO.WaterInput[FTN8] < 32000 THEN				//test the FB for limit - assumes 32767 is max of 10 VDC
					GVL_IO.WaterMotorFwd[FTN8] := TRUE;				// turn on the advance output
					GVL_IO.WaterMotorRvs[FTN8] := FALSE;
					wCycleCount := wCycleCount + 1;
					IF wCycleCount > wMotorTimeOn THEN				//done with timer?
						GVL_IO.WaterMotorFwd[FTN8] := FALSE;		//turn off outputs
						GVL_IO.WaterMotorRvs[FTN8] := FALSE;
						GVL.mb_Output_Coils[GVL.REALTIME_ADVANCE] := FALSE; // reset the advance boolean
						wCycleCount := 0;					//reset the timer counter						
						//  curr % sweep   curr ticks - min tick allowed      max sweep %            max ticks allowed      min ticks allowed
						GVL.mb_Output_Registers[GVL.SWEEPTRIMONPRESS + Index_offset + (FTN8 * GVL.WORDRUNTIMEGROUPSIZE)]	:= (INT_TO_WORD(GVL_IO.InkInput[FTN8]) - GVL.w_InkInputIntMin[FTN8]) * 
								(GVL.mb_Output_Registers[GVL.MAXSWEEPTRIM]+1) / (GVL.w_InkInputIntMax[FTN8] - GVL.w_InkInputIntMin[FTN8]);
						//need the onpress setting pointed to the current % sweep of the positioner
					END_IF
				END_IF
			END_IF
			IF GVL.mb_Output_Coils[GVL.REALTIME_RETARD] THEN
				IF GVL_IO.WaterInput[FTN8] > 800 THEN				//test the FB for limit - assumes 32767 is max of 10 VDC
					GVL_IO.WaterMotorFwd[FTN8] := FALSE;				// turn on the reverse output
					GVL_IO.WaterMotorRvs[FTN8] := TRUE;
					wCycleCount := wCycleCount + 1;
					IF wCycleCount > wMotorTimeOn THEN				//done with timer?
						GVL_IO.WaterMotorFwd[FTN8] := FALSE;		//turn off outputs
						GVL_IO.WaterMotorRvs[FTN8] := FALSE;
						GVL.mb_Output_Coils[GVL.REALTIME_RETARD] := FALSE; // reset the reverse boolean
						wCycleCount := 0;					//reset the timer counter						
						//  curr % sweep   curr ticks - min tick allowed      max sweep %            max ticks allowed      min ticks allowed
						GVL.mb_Output_Registers[GVL.SWEEPTRIMONPRESS + Index_offset + (FTN8 * GVL.WORDRUNTIMEGROUPSIZE)]	:= (INT_TO_WORD(GVL_IO.InkInput[FTN8]) - GVL.w_InkInputIntMin[FTN8]) * 
								(GVL.mb_Output_Registers[GVL.MAXSWEEPTRIM]+1) / (GVL.w_InkInputIntMax[FTN8] - GVL.w_InkInputIntMin[FTN8]);
						//need the onpress setting pointed to the current % sweep of the positioner
					END_IF
				END_IF
			END_IF
		GVL.SWPWTR_OUTPUT:
			IF( GVL.b_DINTInput) THEN									//how big should the adv / ret control increment be?
				w_output_incr :=  DINT_TO_INT(GVL.d_DINT10V / 100);
			ELSE
				w_output_incr := (GVL.i_INT10V / 100);
			END_IF
			GVL.mb_Output_Registers[GVL.REALTIME_PLC_A2D] :=	INT_TO_WORD(GVL_IO.WaterSweepOut[FTN8]);
			IF GVL.mb_Output_Coils[GVL.REALTIME_ADVANCE] THEN
				IF GVL_IO.WaterSweepOut[FTN8] < (w_output_incr * 100) THEN
					GVL_IO.WaterSweepOut[FTN8] := GVL_IO.WaterSweepOut[FTN8] + w_output_incr;
				END_IF
				GVL.mb_Output_Coils[GVL.REALTIME_ADVANCE] := FALSE;
			END_IF
			IF GVL.mb_Output_Coils[GVL.REALTIME_RETARD] THEN
				IF GVL_IO.WaterSweepOut[FTN8] > w_output_incr THEN
					GVL_IO.WaterSweepOut[FTN8] := GVL_IO.WaterSweepOut[FTN8] - w_output_incr;
				END_IF
				GVL.mb_Output_Coils[GVL.REALTIME_RETARD] := FALSE;
			END_IF			
		END_CASE
	 19:CASE GVL.mb_Output_Registers[GVL.WATERHARDWARETYPE] OF
		GVL.SWPWTR_TIME:
			//GVL.mb_Output_Registers[GVL.REALTIME_PLC_A2D] :=	0;	//nothing to read with FB circuit, just move motor
			IF GVL.mb_Output_Coils[GVL.REALTIME_ADVANCE] THEN		//move the motor forward
				IF TRUE THEN							//test the FB for limit - can't do this, pass through
					GVL_IO.WaterMotorFwd[FTN9] := TRUE;				// turn on the advance output
					GVL_IO.WaterMotorRvs[FTN9] := FALSE;
					wCycleCount := wCycleCount + 1;
					IF wCycleCount > wMotorTimeOn THEN				//done with timer?
						GVL_IO.WaterMotorFwd[FTN9] := FALSE;		//turn off outputs
						GVL_IO.WaterMotorRvs[FTN9] := FALSE;
						GVL.mb_Output_Coils[GVL.REALTIME_ADVANCE] := FALSE; // reset the advance boolean
						wCycleCount := 0;					//reset the timer counter						
					END_IF
				END_IF
			END_IF
			IF GVL.mb_Output_Coils[GVL.REALTIME_RETARD] THEN
				IF TRUE THEN							//test the FB for limit - can't do this, pass through
					GVL_IO.WaterMotorFwd[FTN9] := FALSE;				// turn on the reverse output
					GVL_IO.WaterMotorRvs[FTN9] := TRUE;
					wCycleCount := wCycleCount + 1;
					IF wCycleCount > wMotorTimeOn THEN				//done with timer?
						GVL_IO.WaterMotorFwd[FTN9] := FALSE;		//turn off outputs
						GVL_IO.WaterMotorRvs[FTN9] := FALSE;
						GVL.mb_Output_Coils[GVL.REALTIME_RETARD] := FALSE; // reset the reverse boolean
						wCycleCount := 0;					//reset the timer counter						
					END_IF
				END_IF
			END_IF
		GVL.SWPWTR_FB:
			GVL.mb_Output_Registers[GVL.REALTIME_PLC_A2D] :=	INT_TO_WORD(GVL_IO.WaterInput[FTN9]);
			IF GVL.mb_Output_Coils[GVL.REALTIME_ADVANCE] THEN		//move the motor forward
				IF GVL_IO.WaterInput[FTN9] < 32000 THEN				//test the FB for limit - assumes 32767 is max of 10 VDC
					GVL_IO.WaterMotorFwd[FTN9] := TRUE;				// turn on the advance output
					GVL_IO.WaterMotorRvs[FTN9] := FALSE;
					wCycleCount := wCycleCount + 1;
					IF wCycleCount > wMotorTimeOn THEN				//done with timer?
						GVL_IO.WaterMotorFwd[FTN9] := FALSE;		//turn off outputs
						GVL_IO.WaterMotorRvs[FTN9] := FALSE;
						GVL.mb_Output_Coils[GVL.REALTIME_ADVANCE] := FALSE; // reset the advance boolean
						wCycleCount := 0;					//reset the timer counter						
						//  curr % sweep   curr ticks - min tick allowed      max sweep %            max ticks allowed      min ticks allowed
						GVL.mb_Output_Registers[GVL.SWEEPTRIMONPRESS + Index_offset + (FTN9 * GVL.WORDRUNTIMEGROUPSIZE)]	:= (INT_TO_WORD(GVL_IO.InkInput[FTN9]) - GVL.w_InkInputIntMin[FTN9]) * 
								(GVL.mb_Output_Registers[GVL.MAXSWEEPTRIM]+1) / (GVL.w_InkInputIntMax[FTN9] - GVL.w_InkInputIntMin[FTN9]);
						//need the onpress setting pointed to the current % sweep of the positioner
					END_IF
				END_IF
			END_IF
			IF GVL.mb_Output_Coils[GVL.REALTIME_RETARD] THEN
				IF GVL_IO.WaterInput[FTN9] > 800 THEN				//test the FB for limit - assumes 32767 is max of 10 VDC
					GVL_IO.WaterMotorFwd[FTN9] := FALSE;				// turn on the reverse output
					GVL_IO.WaterMotorRvs[FTN9] := TRUE;
					wCycleCount := wCycleCount + 1;
					IF wCycleCount > wMotorTimeOn THEN				//done with timer?
						GVL_IO.WaterMotorFwd[FTN9] := FALSE;		//turn off outputs
						GVL_IO.WaterMotorRvs[FTN9] := FALSE;
						GVL.mb_Output_Coils[GVL.REALTIME_RETARD] := FALSE; // reset the reverse boolean
						wCycleCount := 0;					//reset the timer counter						
						//  curr % sweep   curr ticks - min tick allowed      max sweep %            max ticks allowed      min ticks allowed
						GVL.mb_Output_Registers[GVL.SWEEPTRIMONPRESS + Index_offset + (FTN9 * GVL.WORDRUNTIMEGROUPSIZE)]	:= (INT_TO_WORD(GVL_IO.InkInput[FTN9]) - GVL.w_InkInputIntMin[FTN9]) * 
								(GVL.mb_Output_Registers[GVL.MAXSWEEPTRIM]+1) / (GVL.w_InkInputIntMax[FTN9] - GVL.w_InkInputIntMin[FTN9]);
						//need the onpress setting pointed to the current % sweep of the positioner
					END_IF
				END_IF
			END_IF
		GVL.SWPWTR_OUTPUT:
			IF( GVL.b_DINTInput) THEN									//how big should the adv / ret control increment be?
				w_output_incr :=  DINT_TO_INT(GVL.d_DINT10V / 100);
			ELSE
				w_output_incr := (GVL.i_INT10V / 100);
			END_IF
			GVL.mb_Output_Registers[GVL.REALTIME_PLC_A2D] :=	INT_TO_WORD(GVL_IO.WaterSweepOut[FTN9]);
			IF GVL.mb_Output_Coils[GVL.REALTIME_ADVANCE] THEN
				IF GVL_IO.WaterSweepOut[FTN9] < (w_output_incr * 100) THEN
					GVL_IO.WaterSweepOut[FTN9] := GVL_IO.WaterSweepOut[FTN9] + w_output_incr;
				END_IF
				GVL.mb_Output_Coils[GVL.REALTIME_ADVANCE] := FALSE;
			END_IF
			IF GVL.mb_Output_Coils[GVL.REALTIME_RETARD] THEN
				IF GVL_IO.WaterSweepOut[FTN9] > w_output_incr THEN
					GVL_IO.WaterSweepOut[FTN9] := GVL_IO.WaterSweepOut[FTN9] - w_output_incr;
				END_IF
				GVL.mb_Output_Coils[GVL.REALTIME_RETARD] := FALSE;
			END_IF			
		END_CASE
	 20:CASE GVL.mb_Output_Registers[GVL.WATERHARDWARETYPE] OF
		GVL.SWPWTR_TIME:
			//GVL.mb_Output_Registers[GVL.REALTIME_PLC_A2D] :=	0;	//nothing to read with FB circuit, just move motor
			IF GVL.mb_Output_Coils[GVL.REALTIME_ADVANCE] THEN		//move the motor forward
				IF TRUE THEN							//test the FB for limit - can't do this, pass through
					GVL_IO.WaterMotorFwd[FTN10] := TRUE;				// turn on the advance output
					GVL_IO.WaterMotorRvs[FTN10] := FALSE;
					wCycleCount := wCycleCount + 1;
					IF wCycleCount > wMotorTimeOn THEN				//done with timer?
						GVL_IO.WaterMotorFwd[FTN10] := FALSE;		//turn off outputs
						GVL_IO.WaterMotorRvs[FTN10] := FALSE;
						GVL.mb_Output_Coils[GVL.REALTIME_ADVANCE] := FALSE; // reset the advance boolean
						wCycleCount := 0;					//reset the timer counter						
					END_IF
				END_IF
			END_IF
			IF GVL.mb_Output_Coils[GVL.REALTIME_RETARD] THEN
				IF TRUE THEN							//test the FB for limit - can't do this, pass through
					GVL_IO.WaterMotorFwd[FTN10] := FALSE;				// turn on the reverse output
					GVL_IO.WaterMotorRvs[FTN10] := TRUE;
					wCycleCount := wCycleCount + 1;
					IF wCycleCount > wMotorTimeOn THEN				//done with timer?
						GVL_IO.WaterMotorFwd[FTN10] := FALSE;		//turn off outputs
						GVL_IO.WaterMotorRvs[FTN10] := FALSE;
						GVL.mb_Output_Coils[GVL.REALTIME_RETARD] := FALSE; // reset the reverse boolean
						wCycleCount := 0;					//reset the timer counter						
					END_IF
				END_IF
			END_IF
		GVL.SWPWTR_FB:
			GVL.mb_Output_Registers[GVL.REALTIME_PLC_A2D] :=	INT_TO_WORD(GVL_IO.WaterInput[FTN10]);
			IF GVL.mb_Output_Coils[GVL.REALTIME_ADVANCE] THEN		//move the motor forward
				IF GVL_IO.WaterInput[FTN10] < 32000 THEN				//test the FB for limit - assumes 32767 is max of 10 VDC
					GVL_IO.WaterMotorFwd[FTN10] := TRUE;				// turn on the advance output
					GVL_IO.WaterMotorRvs[FTN10] := FALSE;
					wCycleCount := wCycleCount + 1;
					IF wCycleCount > wMotorTimeOn THEN				//done with timer?
						GVL_IO.WaterMotorFwd[FTN10] := FALSE;		//turn off outputs
						GVL_IO.WaterMotorRvs[FTN10] := FALSE;
						GVL.mb_Output_Coils[GVL.REALTIME_ADVANCE] := FALSE; // reset the advance boolean
						wCycleCount := 0;					//reset the timer counter						
						//  curr % sweep   curr ticks - min tick allowed      max sweep %            max ticks allowed      min ticks allowed
						GVL.mb_Output_Registers[GVL.SWEEPTRIMONPRESS + Index_offset + (FTN10 * GVL.WORDRUNTIMEGROUPSIZE)]	:= (INT_TO_WORD(GVL_IO.InkInput[FTN10]) - GVL.w_InkInputIntMin[FTN10]) * 
								(GVL.mb_Output_Registers[GVL.MAXSWEEPTRIM]+1) / (GVL.w_InkInputIntMax[FTN10] - GVL.w_InkInputIntMin[FTN10]);
						//need the onpress setting pointed to the current % sweep of the positioner
					END_IF
				END_IF
			END_IF
			IF GVL.mb_Output_Coils[GVL.REALTIME_RETARD] THEN
				IF GVL_IO.WaterInput[FTN10] > 800 THEN				//test the FB for limit - assumes 32767 is max of 10 VDC
					GVL_IO.WaterMotorFwd[FTN10] := FALSE;				// turn on the reverse output
					GVL_IO.WaterMotorRvs[FTN10] := TRUE;
					wCycleCount := wCycleCount + 1;
					IF wCycleCount > wMotorTimeOn THEN				//done with timer?
						GVL_IO.WaterMotorFwd[FTN10] := FALSE;		//turn off outputs
						GVL_IO.WaterMotorRvs[FTN10] := FALSE;
						GVL.mb_Output_Coils[GVL.REALTIME_RETARD] := FALSE; // reset the reverse boolean
						wCycleCount := 0;					//reset the timer counter						
						//  curr % sweep   curr ticks - min tick allowed      max sweep %            max ticks allowed      min ticks allowed
						GVL.mb_Output_Registers[GVL.SWEEPTRIMONPRESS + Index_offset + (FTN10 * GVL.WORDRUNTIMEGROUPSIZE)]	:= (INT_TO_WORD(GVL_IO.InkInput[FTN10]) - GVL.w_InkInputIntMin[FTN10]) * 
								(GVL.mb_Output_Registers[GVL.MAXSWEEPTRIM]+1) / (GVL.w_InkInputIntMax[FTN10] - GVL.w_InkInputIntMin[FTN10]);
						//need the onpress setting pointed to the current % sweep of the positioner
					END_IF
				END_IF
			END_IF
		GVL.SWPWTR_OUTPUT:
			IF( GVL.b_DINTInput) THEN									//how big should the adv / ret control increment be?
				w_output_incr :=  DINT_TO_INT(GVL.d_DINT10V / 100);
			ELSE
				w_output_incr := (GVL.i_INT10V / 100);
			END_IF
			GVL.mb_Output_Registers[GVL.REALTIME_PLC_A2D] :=	INT_TO_WORD(GVL_IO.WaterSweepOut[FTN10]);
			IF GVL.mb_Output_Coils[GVL.REALTIME_ADVANCE] THEN
				IF GVL_IO.WaterSweepOut[FTN10] < (w_output_incr * 100) THEN
					GVL_IO.WaterSweepOut[FTN10] := GVL_IO.WaterSweepOut[FTN10] + w_output_incr;
				END_IF
				GVL.mb_Output_Coils[GVL.REALTIME_ADVANCE] := FALSE;
			END_IF
			IF GVL.mb_Output_Coils[GVL.REALTIME_RETARD] THEN
				IF GVL_IO.WaterSweepOut[FTN10] > w_output_incr THEN
					GVL_IO.WaterSweepOut[FTN10] := GVL_IO.WaterSweepOut[FTN10] - w_output_incr;
				END_IF
				GVL.mb_Output_Coils[GVL.REALTIME_RETARD] := FALSE;
			END_IF			
		END_CASE
	 21:   							//press speed analog monitoring
		IF (GVL.b_DINTInput) THEN 
			GVL.mb_Output_Registers[GVL.REALTIME_PLC_A2D] :=	DINT_TO_WORD(GVL_IO.d_PressSpeed/(GVL.d_DINT10V/GVL.i_INT10V))*10;	//press speed (int type)
		ELSE
			GVL.mb_Output_Registers[GVL.REALTIME_PLC_A2D] :=	INT_TO_WORD(GVL_IO.i_PressSpeed);	//press speed (int type)
		END_IF
		GVL.mb_Output_Coils[GVL.REALTIME_ADVANCE] := FALSE; // reset the advance boolean - no adjustment possible here
		GVL.mb_Output_Coils[GVL.REALTIME_RETARD] := FALSE; // reset the reverse boolean
	 22:	//Circ FB Ftn 1
			GVL.mb_Output_Registers[GVL.REALTIME_PLC_A2D] :=	INT_TO_WORD(GVL_IO.CircMotorPot[FTN1]);
			w_temp_index	:= GVL.RUNREG_START+(GVL.RUNREG_SIZE*3*FTN1)+(GVL.RUNREG_SIZE*GVL.iCIRC);
			IF GVL.mb_Output_Coils[GVL.REALTIME_ADVANCE] THEN		//move the motor forward
				IF GVL_IO.CircMotorPot[FTN1] < 32000 THEN				//test the FB for limit - assumes 32767 is max of 10 VDC
					GVL_IO.CircMotorRelay[FTN1,GVL.iPlus] := TRUE;				// turn on the advance output
					GVL_IO.CircMotorRelay[FTN1,GVL.iMinus] := FALSE;
					wCycleCount := wCycleCount + 1;
					IF (wCycleCount > wMotorTimeOn) OR GVL_IO.CircMotorLimit[FTN1,GVL.iPlus] OR
							GVL_IO.CircMotorLimit[FTN1,GVL.iMinus] THEN	//done with timer or any limit activated
						GVL_IO.CircMotorRelay[FTN1,GVL.iPlus] := FALSE;		//turn off outputs
						GVL_IO.CircMotorRelay[FTN1,GVL.iMinus] := FALSE;
						GVL.mb_Output_Coils[GVL.REALTIME_ADVANCE] := FALSE; // reset the advance boolean
						wCycleCount := 0;					//reset the timer counter						
						nRawFBpos	:=	GVL_IO.CircMotorPot[FTN1];
						nActualPos		:= 	LREAL_TO_DINT(
							INT_TO_LREAL(GVL.w_RegisterConfig[Index,GVL.iCIRC,0 ]) +						//base is min position
							(((INT_TO_LREAL(nRawFBpos - GVL.w_RegisterConfig[Index,GVL.iCIRC,2 ])) 			//voltage offset from low calibration
							* 	(INT_TO_LREAL(GVL.w_RegisterConfig[Index,GVL.iCIRC,1 ] - GVL.w_RegisterConfig[Index,GVL.iCIRC,0 ])))	//total position length
							/	( INT_TO_LREAL(GVL.w_RegisterConfig[Index,GVL.iCIRC,3 ] - GVL.w_RegisterConfig[Index,GVL.iCIRC,2 ])))	//total voltage range
							);
						GVL.mb_Output_Registers[w_temp_index+(GVL.iActualPosition)]	:= 
								DINT_TO_WORD(nActualPos);		//post the scaled actual position here to OUTPUT

					END_IF
				END_IF
			END_IF
			IF GVL.mb_Output_Coils[GVL.REALTIME_RETARD] THEN
				IF GVL_IO.CircMotorPot[FTN1] > 800 THEN				//test the FB for limit - assumes 32767 is max of 10 VDC
					GVL_IO.CircMotorRelay[FTN1,GVL.iPlus] := FALSE;				// turn on the reverse output
					GVL_IO.CircMotorRelay[FTN1,GVL.iMinus] := TRUE;
					wCycleCount := wCycleCount + 1;
					IF (wCycleCount > wMotorTimeOn) OR GVL_IO.CircMotorLimit[FTN1,GVL.iPlus] OR
							GVL_IO.CircMotorLimit[FTN1,GVL.iMinus] THEN	//done with timer or any limit activated
						GVL_IO.CircMotorRelay[FTN1,GVL.iPlus] := FALSE;		//turn off outputs
						GVL_IO.CircMotorRelay[FTN1,GVL.iMinus] := FALSE;
						GVL.mb_Output_Coils[GVL.REALTIME_RETARD] := FALSE; // reset the reverse boolean
						wCycleCount := 0;					//reset the timer counter						
						nRawFBpos	:=	GVL_IO.CircMotorPot[FTN1];
						nActualPos		:= 	LREAL_TO_DINT(
							INT_TO_LREAL(GVL.w_RegisterConfig[Index,GVL.iCIRC,0 ]) +						//base is min position
							(((INT_TO_LREAL(nRawFBpos - GVL.w_RegisterConfig[Index,GVL.iCIRC,2 ])) 			//voltage offset from low calibration
							* 	(INT_TO_LREAL(GVL.w_RegisterConfig[Index,GVL.iCIRC,1 ] - GVL.w_RegisterConfig[Index,GVL.iCIRC,0 ])))	//total position length
							/	( INT_TO_LREAL(GVL.w_RegisterConfig[Index,GVL.iCIRC,3 ] - GVL.w_RegisterConfig[Index,GVL.iCIRC,2 ])))	//total voltage range
							);
						GVL.mb_Output_Registers[w_temp_index+(GVL.iActualPosition)]	:= 
								DINT_TO_WORD(nActualPos);		//post the scaled actual position here to OUTPUT
					END_IF
				END_IF
			END_IF
	 23:	//Circ FB Ftn 2
			GVL.mb_Output_Registers[GVL.REALTIME_PLC_A2D] :=	INT_TO_WORD(GVL_IO.CircMotorPot[FTN2]);
			w_temp_index	:= GVL.RUNREG_START+(GVL.RUNREG_SIZE*3*FTN2)+(GVL.RUNREG_SIZE*GVL.iCIRC);
			IF GVL.mb_Output_Coils[GVL.REALTIME_ADVANCE] THEN		//move the motor forward
				IF GVL_IO.CircMotorPot[FTN2] < 32000 THEN				//test the FB for limit - assumes 32767 is max of 10 VDC
					GVL_IO.CircMotorRelay[FTN2,GVL.iPlus] := TRUE;				// turn on the advance output
					GVL_IO.CircMotorRelay[FTN2,GVL.iMinus] := FALSE;
					wCycleCount := wCycleCount + 1;
					IF (wCycleCount > wMotorTimeOn) OR GVL_IO.CircMotorLimit[FTN2,GVL.iPlus] OR
							GVL_IO.CircMotorLimit[FTN2,GVL.iMinus] THEN	//done with timer or any limit activated
						GVL_IO.CircMotorRelay[FTN2,GVL.iPlus] := FALSE;		//turn off outputs
						GVL_IO.CircMotorRelay[FTN2,GVL.iMinus] := FALSE;
						GVL.mb_Output_Coils[GVL.REALTIME_ADVANCE] := FALSE; // reset the advance boolean
						wCycleCount := 0;					//reset the timer counter						
						nRawFBpos	:=	GVL_IO.CircMotorPot[FTN2];
						nActualPos		:= 	LREAL_TO_DINT(
							INT_TO_LREAL(GVL.w_RegisterConfig[Index,GVL.iCIRC,0 ]) +						//base is min position
							(((INT_TO_LREAL(nRawFBpos - GVL.w_RegisterConfig[Index,GVL.iCIRC,2 ])) 			//voltage offset from low calibration
							* 	(INT_TO_LREAL(GVL.w_RegisterConfig[Index,GVL.iCIRC,1 ] - GVL.w_RegisterConfig[Index,GVL.iCIRC,0 ])))	//total position length
							/	( INT_TO_LREAL(GVL.w_RegisterConfig[Index,GVL.iCIRC,3 ] - GVL.w_RegisterConfig[Index,GVL.iCIRC,2 ])))	//total voltage range
							);
						GVL.mb_Output_Registers[w_temp_index+(GVL.iActualPosition)]	:= 
								DINT_TO_WORD(nActualPos);		//post the scaled actual position here to OUTPUT

					END_IF
				END_IF
			END_IF
			IF GVL.mb_Output_Coils[GVL.REALTIME_RETARD] THEN
				IF GVL_IO.CircMotorPot[FTN2] > 800 THEN				//test the FB for limit - assumes 32767 is max of 10 VDC
					GVL_IO.CircMotorRelay[FTN2,GVL.iPlus] := FALSE;				// turn on the reverse output
					GVL_IO.CircMotorRelay[FTN2,GVL.iMinus] := TRUE;
					wCycleCount := wCycleCount + 1;
					IF (wCycleCount > wMotorTimeOn) OR GVL_IO.CircMotorLimit[FTN2,GVL.iPlus] OR
							GVL_IO.CircMotorLimit[FTN2,GVL.iMinus] THEN	//done with timer or any limit activated
						GVL_IO.CircMotorRelay[FTN2,GVL.iPlus] := FALSE;		//turn off outputs
						GVL_IO.CircMotorRelay[FTN2,GVL.iMinus] := FALSE;
						GVL.mb_Output_Coils[GVL.REALTIME_RETARD] := FALSE; // reset the reverse boolean
						wCycleCount := 0;					//reset the timer counter						
						nRawFBpos	:=	GVL_IO.CircMotorPot[FTN2];
						nActualPos		:= 	LREAL_TO_DINT(
							INT_TO_LREAL(GVL.w_RegisterConfig[Index,GVL.iCIRC,0 ]) +						//base is min position
							(((INT_TO_LREAL(nRawFBpos - GVL.w_RegisterConfig[Index,GVL.iCIRC,2 ])) 			//voltage offset from low calibration
							* 	(INT_TO_LREAL(GVL.w_RegisterConfig[Index,GVL.iCIRC,1 ] - GVL.w_RegisterConfig[Index,GVL.iCIRC,0 ])))	//total position length
							/	( INT_TO_LREAL(GVL.w_RegisterConfig[Index,GVL.iCIRC,3 ] - GVL.w_RegisterConfig[Index,GVL.iCIRC,2 ])))	//total voltage range
							);
						GVL.mb_Output_Registers[w_temp_index+(GVL.iActualPosition)]	:= 
								DINT_TO_WORD(nActualPos);		//post the scaled actual position here to OUTPUT
					END_IF
				END_IF
			END_IF
	 24:	//Circ FB Ftn 3
			GVL.mb_Output_Registers[GVL.REALTIME_PLC_A2D] :=	INT_TO_WORD(GVL_IO.CircMotorPot[FTN3]);
			w_temp_index	:= GVL.RUNREG_START+(GVL.RUNREG_SIZE*3*FTN3)+(GVL.RUNREG_SIZE*GVL.iCIRC);
			IF GVL.mb_Output_Coils[GVL.REALTIME_ADVANCE] THEN		//move the motor forward
				IF GVL_IO.CircMotorPot[FTN3] < 32000 THEN				//test the FB for limit - assumes 32767 is max of 10 VDC
					GVL_IO.CircMotorRelay[FTN3,GVL.iPlus] := TRUE;				// turn on the advance output
					GVL_IO.CircMotorRelay[FTN3,GVL.iMinus] := FALSE;
					wCycleCount := wCycleCount + 1;
					IF (wCycleCount > wMotorTimeOn) OR GVL_IO.CircMotorLimit[FTN3,GVL.iPlus] OR
							GVL_IO.CircMotorLimit[FTN3,GVL.iMinus] THEN	//done with timer or any limit activated
						GVL_IO.CircMotorRelay[FTN3,GVL.iPlus] := FALSE;		//turn off outputs
						GVL_IO.CircMotorRelay[FTN3,GVL.iMinus] := FALSE;
						GVL.mb_Output_Coils[GVL.REALTIME_ADVANCE] := FALSE; // reset the advance boolean
						wCycleCount := 0;					//reset the timer counter						
						nRawFBpos	:=	GVL_IO.CircMotorPot[FTN3];
						nActualPos		:= 	LREAL_TO_DINT(
							INT_TO_LREAL(GVL.w_RegisterConfig[Index,GVL.iCIRC,0 ]) +						//base is min position
							(((INT_TO_LREAL(nRawFBpos - GVL.w_RegisterConfig[Index,GVL.iCIRC,2 ])) 			//voltage offset from low calibration
							* 	(INT_TO_LREAL(GVL.w_RegisterConfig[Index,GVL.iCIRC,1 ] - GVL.w_RegisterConfig[Index,GVL.iCIRC,0 ])))	//total position length
							/	( INT_TO_LREAL(GVL.w_RegisterConfig[Index,GVL.iCIRC,3 ] - GVL.w_RegisterConfig[Index,GVL.iCIRC,2 ])))	//total voltage range
							);
						GVL.mb_Output_Registers[w_temp_index+(GVL.iActualPosition)]	:= 
								DINT_TO_WORD(nActualPos);		//post the scaled actual position here to OUTPUT

					END_IF
				END_IF
			END_IF
			IF GVL.mb_Output_Coils[GVL.REALTIME_RETARD] THEN
				IF GVL_IO.CircMotorPot[FTN3] > 800 THEN				//test the FB for limit - assumes 32767 is max of 10 VDC
					GVL_IO.CircMotorRelay[FTN3,GVL.iPlus] := FALSE;				// turn on the reverse output
					GVL_IO.CircMotorRelay[FTN3,GVL.iMinus] := TRUE;
					wCycleCount := wCycleCount + 1;
					IF (wCycleCount > wMotorTimeOn) OR GVL_IO.CircMotorLimit[FTN3,GVL.iPlus] OR
							GVL_IO.CircMotorLimit[FTN3,GVL.iMinus] THEN	//done with timer or any limit activated
						GVL_IO.CircMotorRelay[FTN3,GVL.iPlus] := FALSE;		//turn off outputs
						GVL_IO.CircMotorRelay[FTN3,GVL.iMinus] := FALSE;
						GVL.mb_Output_Coils[GVL.REALTIME_RETARD] := FALSE; // reset the reverse boolean
						wCycleCount := 0;					//reset the timer counter						
						nRawFBpos	:=	GVL_IO.CircMotorPot[FTN3];
						nActualPos		:= 	LREAL_TO_DINT(
							INT_TO_LREAL(GVL.w_RegisterConfig[Index,GVL.iCIRC,0 ]) +						//base is min position
							(((INT_TO_LREAL(nRawFBpos - GVL.w_RegisterConfig[Index,GVL.iCIRC,2 ])) 			//voltage offset from low calibration
							* 	(INT_TO_LREAL(GVL.w_RegisterConfig[Index,GVL.iCIRC,1 ] - GVL.w_RegisterConfig[Index,GVL.iCIRC,0 ])))	//total position length
							/	( INT_TO_LREAL(GVL.w_RegisterConfig[Index,GVL.iCIRC,3 ] - GVL.w_RegisterConfig[Index,GVL.iCIRC,2 ])))	//total voltage range
							);
						GVL.mb_Output_Registers[w_temp_index+(GVL.iActualPosition)]	:= 
								DINT_TO_WORD(nActualPos);		//post the scaled actual position here to OUTPUT
					END_IF
				END_IF
			END_IF
	 25:	//Circ FB Ftn 4
			GVL.mb_Output_Registers[GVL.REALTIME_PLC_A2D] :=	INT_TO_WORD(GVL_IO.CircMotorPot[FTN4]);
			w_temp_index	:= GVL.RUNREG_START+(GVL.RUNREG_SIZE*3*FTN4)+(GVL.RUNREG_SIZE*GVL.iCIRC);
			IF GVL.mb_Output_Coils[GVL.REALTIME_ADVANCE] THEN		//move the motor forward
				IF GVL_IO.CircMotorPot[FTN4] < 32000 THEN				//test the FB for limit - assumes 32767 is max of 10 VDC
					GVL_IO.CircMotorRelay[FTN4,GVL.iPlus] := TRUE;				// turn on the advance output
					GVL_IO.CircMotorRelay[FTN4,GVL.iMinus] := FALSE;
					wCycleCount := wCycleCount + 1;
					IF (wCycleCount > wMotorTimeOn) OR GVL_IO.CircMotorLimit[FTN4,GVL.iPlus] OR
							GVL_IO.CircMotorLimit[FTN4,GVL.iMinus] THEN	//done with timer or any limit activated
						GVL_IO.CircMotorRelay[FTN4,GVL.iPlus] := FALSE;		//turn off outputs
						GVL_IO.CircMotorRelay[FTN4,GVL.iMinus] := FALSE;
						GVL.mb_Output_Coils[GVL.REALTIME_ADVANCE] := FALSE; // reset the advance boolean
						wCycleCount := 0;					//reset the timer counter						
						nRawFBpos	:=	GVL_IO.CircMotorPot[FTN4];
						nActualPos		:= 	LREAL_TO_DINT(
							INT_TO_LREAL(GVL.w_RegisterConfig[Index,GVL.iCIRC,0 ]) +						//base is min position
							(((INT_TO_LREAL(nRawFBpos - GVL.w_RegisterConfig[Index,GVL.iCIRC,2 ])) 			//voltage offset from low calibration
							* 	(INT_TO_LREAL(GVL.w_RegisterConfig[Index,GVL.iCIRC,1 ] - GVL.w_RegisterConfig[Index,GVL.iCIRC,0 ])))	//total position length
							/	( INT_TO_LREAL(GVL.w_RegisterConfig[Index,GVL.iCIRC,3 ] - GVL.w_RegisterConfig[Index,GVL.iCIRC,2 ])))	//total voltage range
							);
						GVL.mb_Output_Registers[w_temp_index+(GVL.iActualPosition)]	:= 
								DINT_TO_WORD(nActualPos);		//post the scaled actual position here to OUTPUT

					END_IF
				END_IF
			END_IF
			IF GVL.mb_Output_Coils[GVL.REALTIME_RETARD] THEN
				IF GVL_IO.CircMotorPot[FTN4] > 800 THEN				//test the FB for limit - assumes 32767 is max of 10 VDC
					GVL_IO.CircMotorRelay[FTN4,GVL.iPlus] := FALSE;				// turn on the reverse output
					GVL_IO.CircMotorRelay[FTN4,GVL.iMinus] := TRUE;
					wCycleCount := wCycleCount + 1;
					IF (wCycleCount > wMotorTimeOn) OR GVL_IO.CircMotorLimit[FTN4,GVL.iPlus] OR
							GVL_IO.CircMotorLimit[FTN4,GVL.iMinus] THEN	//done with timer or any limit activated
						GVL_IO.CircMotorRelay[FTN4,GVL.iPlus] := FALSE;		//turn off outputs
						GVL_IO.CircMotorRelay[FTN4,GVL.iMinus] := FALSE;
						GVL.mb_Output_Coils[GVL.REALTIME_RETARD] := FALSE; // reset the reverse boolean
						wCycleCount := 0;					//reset the timer counter						
						nRawFBpos	:=	GVL_IO.CircMotorPot[FTN4];
						nActualPos		:= 	LREAL_TO_DINT(
							INT_TO_LREAL(GVL.w_RegisterConfig[Index,GVL.iCIRC,0 ]) +						//base is min position
							(((INT_TO_LREAL(nRawFBpos - GVL.w_RegisterConfig[Index,GVL.iCIRC,2 ])) 			//voltage offset from low calibration
							* 	(INT_TO_LREAL(GVL.w_RegisterConfig[Index,GVL.iCIRC,1 ] - GVL.w_RegisterConfig[Index,GVL.iCIRC,0 ])))	//total position length
							/	( INT_TO_LREAL(GVL.w_RegisterConfig[Index,GVL.iCIRC,3 ] - GVL.w_RegisterConfig[Index,GVL.iCIRC,2 ])))	//total voltage range
							);
						GVL.mb_Output_Registers[w_temp_index+(GVL.iActualPosition)]	:= 
								DINT_TO_WORD(nActualPos);		//post the scaled actual position here to OUTPUT
					END_IF
				END_IF
			END_IF
	 26:	//Circ FB Ftn 5
			GVL.mb_Output_Registers[GVL.REALTIME_PLC_A2D] :=	INT_TO_WORD(GVL_IO.CircMotorPot[FTN5]);
			w_temp_index	:= GVL.RUNREG_START+(GVL.RUNREG_SIZE*3*FTN5)+(GVL.RUNREG_SIZE*GVL.iCIRC);
			IF GVL.mb_Output_Coils[GVL.REALTIME_ADVANCE] THEN		//move the motor forward
				IF GVL_IO.CircMotorPot[FTN5] < 32000 THEN				//test the FB for limit - assumes 32767 is max of 10 VDC
					GVL_IO.CircMotorRelay[FTN5,GVL.iPlus] := TRUE;				// turn on the advance output
					GVL_IO.CircMotorRelay[FTN5,GVL.iMinus] := FALSE;
					wCycleCount := wCycleCount + 1;
					IF (wCycleCount > wMotorTimeOn) OR GVL_IO.CircMotorLimit[FTN5,GVL.iPlus] OR
							GVL_IO.CircMotorLimit[FTN5,GVL.iMinus] THEN	//done with timer or any limit activated
						GVL_IO.CircMotorRelay[FTN5,GVL.iPlus] := FALSE;		//turn off outputs
						GVL_IO.CircMotorRelay[FTN5,GVL.iMinus] := FALSE;
						GVL.mb_Output_Coils[GVL.REALTIME_ADVANCE] := FALSE; // reset the advance boolean
						wCycleCount := 0;					//reset the timer counter						
						nRawFBpos	:=	GVL_IO.CircMotorPot[FTN5];
						nActualPos		:= 	LREAL_TO_DINT(
							INT_TO_LREAL(GVL.w_RegisterConfig[Index,GVL.iCIRC,0 ]) +						//base is min position
							(((INT_TO_LREAL(nRawFBpos - GVL.w_RegisterConfig[Index,GVL.iCIRC,2 ])) 			//voltage offset from low calibration
							* 	(INT_TO_LREAL(GVL.w_RegisterConfig[Index,GVL.iCIRC,1 ] - GVL.w_RegisterConfig[Index,GVL.iCIRC,0 ])))	//total position length
							/	( INT_TO_LREAL(GVL.w_RegisterConfig[Index,GVL.iCIRC,3 ] - GVL.w_RegisterConfig[Index,GVL.iCIRC,2 ])))	//total voltage range
							);
						GVL.mb_Output_Registers[w_temp_index+(GVL.iActualPosition)]	:= 
								DINT_TO_WORD(nActualPos);		//post the scaled actual position here to OUTPUT

					END_IF
				END_IF
			END_IF
			IF GVL.mb_Output_Coils[GVL.REALTIME_RETARD] THEN
				IF GVL_IO.CircMotorPot[FTN5] > 800 THEN				//test the FB for limit - assumes 32767 is max of 10 VDC
					GVL_IO.CircMotorRelay[FTN5,GVL.iPlus] := FALSE;				// turn on the reverse output
					GVL_IO.CircMotorRelay[FTN5,GVL.iMinus] := TRUE;
					wCycleCount := wCycleCount + 1;
					IF (wCycleCount > wMotorTimeOn) OR GVL_IO.CircMotorLimit[FTN5,GVL.iPlus] OR
							GVL_IO.CircMotorLimit[FTN5,GVL.iMinus] THEN	//done with timer or any limit activated
						GVL_IO.CircMotorRelay[FTN5,GVL.iPlus] := FALSE;		//turn off outputs
						GVL_IO.CircMotorRelay[FTN5,GVL.iMinus] := FALSE;
						GVL.mb_Output_Coils[GVL.REALTIME_RETARD] := FALSE; // reset the reverse boolean
						wCycleCount := 0;					//reset the timer counter						
						nRawFBpos	:=	GVL_IO.CircMotorPot[FTN5];
						nActualPos		:= 	LREAL_TO_DINT(
							INT_TO_LREAL(GVL.w_RegisterConfig[Index,GVL.iCIRC,0 ]) +						//base is min position
							(((INT_TO_LREAL(nRawFBpos - GVL.w_RegisterConfig[Index,GVL.iCIRC,2 ])) 			//voltage offset from low calibration
							* 	(INT_TO_LREAL(GVL.w_RegisterConfig[Index,GVL.iCIRC,1 ] - GVL.w_RegisterConfig[Index,GVL.iCIRC,0 ])))	//total position length
							/	( INT_TO_LREAL(GVL.w_RegisterConfig[Index,GVL.iCIRC,3 ] - GVL.w_RegisterConfig[Index,GVL.iCIRC,2 ])))	//total voltage range
							);
						GVL.mb_Output_Registers[w_temp_index+(GVL.iActualPosition)]	:= 
								DINT_TO_WORD(nActualPos);		//post the scaled actual position here to OUTPUT
					END_IF
				END_IF
			END_IF
	 27:	//Circ FB Ftn 6
			GVL.mb_Output_Registers[GVL.REALTIME_PLC_A2D] :=	INT_TO_WORD(GVL_IO.CircMotorPot[FTN6]);
		//	FTN 6 special
			w_temp_index	:= GVL.RUNREG_START+(GVL.RUNREG_SIZE*3*FTN6)+(GVL.RUNREG_SIZE*GVL.iCIRC)+10;
			IF GVL.mb_Output_Coils[GVL.REALTIME_ADVANCE] THEN		//move the motor forward
				IF GVL_IO.CircMotorPot[FTN6] < 32000 THEN				//test the FB for limit - assumes 32767 is max of 10 VDC
					GVL_IO.CircMotorRelay[FTN6,GVL.iPlus] := TRUE;				// turn on the advance output
					GVL_IO.CircMotorRelay[FTN6,GVL.iMinus] := FALSE;
					wCycleCount := wCycleCount + 1;
					IF (wCycleCount > wMotorTimeOn) OR GVL_IO.CircMotorLimit[FTN6,GVL.iPlus] OR
							GVL_IO.CircMotorLimit[FTN6,GVL.iMinus] THEN	//done with timer or any limit activated
						GVL_IO.CircMotorRelay[FTN6,GVL.iPlus] := FALSE;		//turn off outputs
						GVL_IO.CircMotorRelay[FTN6,GVL.iMinus] := FALSE;
						GVL.mb_Output_Coils[GVL.REALTIME_ADVANCE] := FALSE; // reset the advance boolean
						wCycleCount := 0;					//reset the timer counter						
						nRawFBpos	:=	GVL_IO.CircMotorPot[FTN6];
						nActualPos		:= 	LREAL_TO_DINT(
							INT_TO_LREAL(GVL.w_RegisterConfig[Index,GVL.iCIRC,0 ]) +						//base is min position
							(((INT_TO_LREAL(nRawFBpos - GVL.w_RegisterConfig[Index,GVL.iCIRC,2 ])) 			//voltage offset from low calibration
							* 	(INT_TO_LREAL(GVL.w_RegisterConfig[Index,GVL.iCIRC,1 ] - GVL.w_RegisterConfig[Index,GVL.iCIRC,0 ])))	//total position length
							/	( INT_TO_LREAL(GVL.w_RegisterConfig[Index,GVL.iCIRC,3 ] - GVL.w_RegisterConfig[Index,GVL.iCIRC,2 ])))	//total voltage range
							);
						GVL.mb_Output_Registers[w_temp_index+(GVL.iActualPosition)]	:= 
								DINT_TO_WORD(nActualPos);		//post the scaled actual position here to OUTPUT

					END_IF
				END_IF
			END_IF
			IF GVL.mb_Output_Coils[GVL.REALTIME_RETARD] THEN
				IF GVL_IO.CircMotorPot[FTN6] > 800 THEN				//test the FB for limit - assumes 32767 is max of 10 VDC
					GVL_IO.CircMotorRelay[FTN6,GVL.iPlus] := FALSE;				// turn on the reverse output
					GVL_IO.CircMotorRelay[FTN6,GVL.iMinus] := TRUE;
					wCycleCount := wCycleCount + 1;
					IF (wCycleCount > wMotorTimeOn) OR GVL_IO.CircMotorLimit[FTN6,GVL.iPlus] OR
							GVL_IO.CircMotorLimit[FTN6,GVL.iMinus] THEN	//done with timer or any limit activated
						GVL_IO.CircMotorRelay[FTN6,GVL.iPlus] := FALSE;		//turn off outputs
						GVL_IO.CircMotorRelay[FTN6,GVL.iMinus] := FALSE;
						GVL.mb_Output_Coils[GVL.REALTIME_RETARD] := FALSE; // reset the reverse boolean
						wCycleCount := 0;					//reset the timer counter						
						nRawFBpos	:=	GVL_IO.CircMotorPot[FTN6];
						nActualPos		:= 	LREAL_TO_DINT(
							INT_TO_LREAL(GVL.w_RegisterConfig[Index,GVL.iCIRC,0 ]) +						//base is min position
							(((INT_TO_LREAL(nRawFBpos - GVL.w_RegisterConfig[Index,GVL.iCIRC,2 ])) 			//voltage offset from low calibration
							* 	(INT_TO_LREAL(GVL.w_RegisterConfig[Index,GVL.iCIRC,1 ] - GVL.w_RegisterConfig[Index,GVL.iCIRC,0 ])))	//total position length
							/	( INT_TO_LREAL(GVL.w_RegisterConfig[Index,GVL.iCIRC,3 ] - GVL.w_RegisterConfig[Index,GVL.iCIRC,2 ])))	//total voltage range
							);
						GVL.mb_Output_Registers[w_temp_index+(GVL.iActualPosition)]	:= 
								DINT_TO_WORD(nActualPos);		//post the scaled actual position here to OUTPUT
					END_IF
				END_IF
			END_IF
	 28:	//Circ FB Ftn 7
			GVL.mb_Output_Registers[GVL.REALTIME_PLC_A2D] :=	INT_TO_WORD(GVL_IO.CircMotorPot[FTN7]);
			w_temp_index	:= GVL.RUNREG_START+(GVL.RUNREG_SIZE*3*FTN7)+(GVL.RUNREG_SIZE*GVL.iCIRC)+10;
			IF GVL.mb_Output_Coils[GVL.REALTIME_ADVANCE] THEN		//move the motor forward
				IF GVL_IO.CircMotorPot[FTN7] < 32000 THEN				//test the FB for limit - assumes 32767 is max of 10 VDC
					GVL_IO.CircMotorRelay[FTN7,GVL.iPlus] := TRUE;				// turn on the advance output
					GVL_IO.CircMotorRelay[FTN7,GVL.iMinus] := FALSE;
					wCycleCount := wCycleCount + 1;
					IF (wCycleCount > wMotorTimeOn) OR GVL_IO.CircMotorLimit[FTN7,GVL.iPlus] OR
							GVL_IO.CircMotorLimit[FTN7,GVL.iMinus] THEN	//done with timer or any limit activated
						GVL_IO.CircMotorRelay[FTN7,GVL.iPlus] := FALSE;		//turn off outputs
						GVL_IO.CircMotorRelay[FTN7,GVL.iMinus] := FALSE;
						GVL.mb_Output_Coils[GVL.REALTIME_ADVANCE] := FALSE; // reset the advance boolean
						wCycleCount := 0;					//reset the timer counter						
						nRawFBpos	:=	GVL_IO.CircMotorPot[FTN7];
						nActualPos		:= 	LREAL_TO_DINT(
							INT_TO_LREAL(GVL.w_RegisterConfig[Index,GVL.iCIRC,0 ]) +						//base is min position
							(((INT_TO_LREAL(nRawFBpos - GVL.w_RegisterConfig[Index,GVL.iCIRC,2 ])) 			//voltage offset from low calibration
							* 	(INT_TO_LREAL(GVL.w_RegisterConfig[Index,GVL.iCIRC,1 ] - GVL.w_RegisterConfig[Index,GVL.iCIRC,0 ])))	//total position length
							/	( INT_TO_LREAL(GVL.w_RegisterConfig[Index,GVL.iCIRC,3 ] - GVL.w_RegisterConfig[Index,GVL.iCIRC,2 ])))	//total voltage range
							);
						GVL.mb_Output_Registers[w_temp_index+(GVL.iActualPosition)]	:= 
								DINT_TO_WORD(nActualPos);		//post the scaled actual position here to OUTPUT

					END_IF
				END_IF
			END_IF
			IF GVL.mb_Output_Coils[GVL.REALTIME_RETARD] THEN
				IF GVL_IO.CircMotorPot[FTN7] > 800 THEN				//test the FB for limit - assumes 32767 is max of 10 VDC
					GVL_IO.CircMotorRelay[FTN7,GVL.iPlus] := FALSE;				// turn on the reverse output
					GVL_IO.CircMotorRelay[FTN7,GVL.iMinus] := TRUE;
					wCycleCount := wCycleCount + 1;
					IF (wCycleCount > wMotorTimeOn) OR GVL_IO.CircMotorLimit[FTN7,GVL.iPlus] OR
							GVL_IO.CircMotorLimit[FTN7,GVL.iMinus] THEN	//done with timer or any limit activated
						GVL_IO.CircMotorRelay[FTN7,GVL.iPlus] := FALSE;		//turn off outputs
						GVL_IO.CircMotorRelay[FTN7,GVL.iMinus] := FALSE;
						GVL.mb_Output_Coils[GVL.REALTIME_RETARD] := FALSE; // reset the reverse boolean
						wCycleCount := 0;					//reset the timer counter						
						nRawFBpos	:=	GVL_IO.CircMotorPot[FTN7];
						nActualPos		:= 	LREAL_TO_DINT(
							INT_TO_LREAL(GVL.w_RegisterConfig[Index,GVL.iCIRC,0 ]) +						//base is min position
							(((INT_TO_LREAL(nRawFBpos - GVL.w_RegisterConfig[Index,GVL.iCIRC,2 ])) 			//voltage offset from low calibration
							* 	(INT_TO_LREAL(GVL.w_RegisterConfig[Index,GVL.iCIRC,1 ] - GVL.w_RegisterConfig[Index,GVL.iCIRC,0 ])))	//total position length
							/	( INT_TO_LREAL(GVL.w_RegisterConfig[Index,GVL.iCIRC,3 ] - GVL.w_RegisterConfig[Index,GVL.iCIRC,2 ])))	//total voltage range
							);
						GVL.mb_Output_Registers[w_temp_index+(GVL.iActualPosition)]	:= 
								DINT_TO_WORD(nActualPos);		//post the scaled actual position here to OUTPUT
					END_IF
				END_IF
			END_IF
	 29:	//Circ FB Ftn 8
			GVL.mb_Output_Registers[GVL.REALTIME_PLC_A2D] :=	INT_TO_WORD(GVL_IO.CircMotorPot[FTN8]);
			w_temp_index	:= GVL.RUNREG_START+(GVL.RUNREG_SIZE*3*FTN8)+(GVL.RUNREG_SIZE*GVL.iCIRC)+10;
			IF GVL.mb_Output_Coils[GVL.REALTIME_ADVANCE] THEN		//move the motor forward
				IF GVL_IO.CircMotorPot[FTN8] < 32000 THEN				//test the FB for limit - assumes 32767 is max of 10 VDC
					GVL_IO.CircMotorRelay[FTN8,GVL.iPlus] := TRUE;				// turn on the advance output
					GVL_IO.CircMotorRelay[FTN8,GVL.iMinus] := FALSE;
					wCycleCount := wCycleCount + 1;
					IF (wCycleCount > wMotorTimeOn) OR GVL_IO.CircMotorLimit[FTN8,GVL.iPlus] OR
							GVL_IO.CircMotorLimit[FTN8,GVL.iMinus] THEN	//done with timer or any limit activated
						GVL_IO.CircMotorRelay[FTN8,GVL.iPlus] := FALSE;		//turn off outputs
						GVL_IO.CircMotorRelay[FTN8,GVL.iMinus] := FALSE;
						GVL.mb_Output_Coils[GVL.REALTIME_ADVANCE] := FALSE; // reset the advance boolean
						wCycleCount := 0;					//reset the timer counter						
						nRawFBpos	:=	GVL_IO.CircMotorPot[FTN8];
						nActualPos		:= 	LREAL_TO_DINT(
							INT_TO_LREAL(GVL.w_RegisterConfig[Index,GVL.iCIRC,0 ]) +						//base is min position
							(((INT_TO_LREAL(nRawFBpos - GVL.w_RegisterConfig[Index,GVL.iCIRC,2 ])) 			//voltage offset from low calibration
							* 	(INT_TO_LREAL(GVL.w_RegisterConfig[Index,GVL.iCIRC,1 ] - GVL.w_RegisterConfig[Index,GVL.iCIRC,0 ])))	//total position length
							/	( INT_TO_LREAL(GVL.w_RegisterConfig[Index,GVL.iCIRC,3 ] - GVL.w_RegisterConfig[Index,GVL.iCIRC,2 ])))	//total voltage range
							);
						GVL.mb_Output_Registers[w_temp_index+(GVL.iActualPosition)]	:= 
								DINT_TO_WORD(nActualPos);		//post the scaled actual position here to OUTPUT

					END_IF
				END_IF
			END_IF
			IF GVL.mb_Output_Coils[GVL.REALTIME_RETARD] THEN
				IF GVL_IO.CircMotorPot[FTN8] > 800 THEN				//test the FB for limit - assumes 32767 is max of 10 VDC
					GVL_IO.CircMotorRelay[FTN8,GVL.iPlus] := FALSE;				// turn on the reverse output
					GVL_IO.CircMotorRelay[FTN8,GVL.iMinus] := TRUE;
					wCycleCount := wCycleCount + 1;
					IF (wCycleCount > wMotorTimeOn) OR GVL_IO.CircMotorLimit[FTN8,GVL.iPlus] OR
							GVL_IO.CircMotorLimit[FTN8,GVL.iMinus] THEN	//done with timer or any limit activated
						GVL_IO.CircMotorRelay[FTN8,GVL.iPlus] := FALSE;		//turn off outputs
						GVL_IO.CircMotorRelay[FTN8,GVL.iMinus] := FALSE;
						GVL.mb_Output_Coils[GVL.REALTIME_RETARD] := FALSE; // reset the reverse boolean
						wCycleCount := 0;					//reset the timer counter						
						nRawFBpos	:=	GVL_IO.CircMotorPot[FTN8];
						nActualPos		:= 	LREAL_TO_DINT(
							INT_TO_LREAL(GVL.w_RegisterConfig[Index,GVL.iCIRC,0 ]) +						//base is min position
							(((INT_TO_LREAL(nRawFBpos - GVL.w_RegisterConfig[Index,GVL.iCIRC,2 ])) 			//voltage offset from low calibration
							* 	(INT_TO_LREAL(GVL.w_RegisterConfig[Index,GVL.iCIRC,1 ] - GVL.w_RegisterConfig[Index,GVL.iCIRC,0 ])))	//total position length
							/	( INT_TO_LREAL(GVL.w_RegisterConfig[Index,GVL.iCIRC,3 ] - GVL.w_RegisterConfig[Index,GVL.iCIRC,2 ])))	//total voltage range
							);
						GVL.mb_Output_Registers[w_temp_index+(GVL.iActualPosition)]	:= 
								DINT_TO_WORD(nActualPos);		//post the scaled actual position here to OUTPUT
					END_IF
				END_IF
			END_IF
	 30:	//Circ FB Ftn 9
			GVL.mb_Output_Registers[GVL.REALTIME_PLC_A2D] :=	INT_TO_WORD(GVL_IO.CircMotorPot[FTN9]);
			w_temp_index	:= GVL.RUNREG_START+(GVL.RUNREG_SIZE*3*FTN9)+(GVL.RUNREG_SIZE*GVL.iCIRC)+10;
			IF GVL.mb_Output_Coils[GVL.REALTIME_ADVANCE] THEN		//move the motor forward
				IF GVL_IO.CircMotorPot[FTN9] < 32000 THEN				//test the FB for limit - assumes 32767 is max of 10 VDC
					GVL_IO.CircMotorRelay[FTN9,GVL.iPlus] := TRUE;				// turn on the advance output
					GVL_IO.CircMotorRelay[FTN9,GVL.iMinus] := FALSE;
					wCycleCount := wCycleCount + 1;
					IF (wCycleCount > wMotorTimeOn) OR GVL_IO.CircMotorLimit[FTN9,GVL.iPlus] OR
							GVL_IO.CircMotorLimit[FTN9,GVL.iMinus] THEN	//done with timer or any limit activated
						GVL_IO.CircMotorRelay[FTN9,GVL.iPlus] := FALSE;		//turn off outputs
						GVL_IO.CircMotorRelay[FTN9,GVL.iMinus] := FALSE;
						GVL.mb_Output_Coils[GVL.REALTIME_ADVANCE] := FALSE; // reset the advance boolean
						wCycleCount := 0;					//reset the timer counter						
						nRawFBpos	:=	GVL_IO.CircMotorPot[FTN9];
						nActualPos		:= 	LREAL_TO_DINT(
							INT_TO_LREAL(GVL.w_RegisterConfig[Index,GVL.iCIRC,0 ]) +						//base is min position
							(((INT_TO_LREAL(nRawFBpos - GVL.w_RegisterConfig[Index,GVL.iCIRC,2 ])) 			//voltage offset from low calibration
							* 	(INT_TO_LREAL(GVL.w_RegisterConfig[Index,GVL.iCIRC,1 ] - GVL.w_RegisterConfig[Index,GVL.iCIRC,0 ])))	//total position length
							/	( INT_TO_LREAL(GVL.w_RegisterConfig[Index,GVL.iCIRC,3 ] - GVL.w_RegisterConfig[Index,GVL.iCIRC,2 ])))	//total voltage range
							);
						GVL.mb_Output_Registers[w_temp_index+(GVL.iActualPosition)]	:= 
								DINT_TO_WORD(nActualPos);		//post the scaled actual position here to OUTPUT

					END_IF
				END_IF
			END_IF
			IF GVL.mb_Output_Coils[GVL.REALTIME_RETARD] THEN
				IF GVL_IO.CircMotorPot[FTN9] > 800 THEN				//test the FB for limit - assumes 32767 is max of 10 VDC
					GVL_IO.CircMotorRelay[FTN9,GVL.iPlus] := FALSE;				// turn on the reverse output
					GVL_IO.CircMotorRelay[FTN9,GVL.iMinus] := TRUE;
					wCycleCount := wCycleCount + 1;
					IF (wCycleCount > wMotorTimeOn) OR GVL_IO.CircMotorLimit[FTN9,GVL.iPlus] OR
							GVL_IO.CircMotorLimit[FTN9,GVL.iMinus] THEN	//done with timer or any limit activated
						GVL_IO.CircMotorRelay[FTN9,GVL.iPlus] := FALSE;		//turn off outputs
						GVL_IO.CircMotorRelay[FTN9,GVL.iMinus] := FALSE;
						GVL.mb_Output_Coils[GVL.REALTIME_RETARD] := FALSE; // reset the reverse boolean
						wCycleCount := 0;					//reset the timer counter						
						nRawFBpos	:=	GVL_IO.CircMotorPot[FTN9];
						nActualPos		:= 	LREAL_TO_DINT(
							INT_TO_LREAL(GVL.w_RegisterConfig[Index,GVL.iCIRC,0 ]) +						//base is min position
							(((INT_TO_LREAL(nRawFBpos - GVL.w_RegisterConfig[Index,GVL.iCIRC,2 ])) 			//voltage offset from low calibration
							* 	(INT_TO_LREAL(GVL.w_RegisterConfig[Index,GVL.iCIRC,1 ] - GVL.w_RegisterConfig[Index,GVL.iCIRC,0 ])))	//total position length
							/	( INT_TO_LREAL(GVL.w_RegisterConfig[Index,GVL.iCIRC,3 ] - GVL.w_RegisterConfig[Index,GVL.iCIRC,2 ])))	//total voltage range
							);
						GVL.mb_Output_Registers[w_temp_index+(GVL.iActualPosition)]	:= 
								DINT_TO_WORD(nActualPos);		//post the scaled actual position here to OUTPUT
					END_IF
				END_IF
			END_IF
	 31:	//Circ FB Ftn 10
			GVL.mb_Output_Registers[GVL.REALTIME_PLC_A2D] :=	INT_TO_WORD(GVL_IO.CircMotorPot[FTN10]);
			w_temp_index	:= GVL.RUNREG_START+(GVL.RUNREG_SIZE*3*FTN10)+(GVL.RUNREG_SIZE*GVL.iCIRC)+10;
			IF GVL.mb_Output_Coils[GVL.REALTIME_ADVANCE] THEN		//move the motor forward
				IF GVL_IO.CircMotorPot[FTN10] < 32000 THEN				//test the FB for limit - assumes 32767 is max of 10 VDC
					GVL_IO.CircMotorRelay[FTN10,GVL.iPlus] := TRUE;				// turn on the advance output
					GVL_IO.CircMotorRelay[FTN10,GVL.iMinus] := FALSE;
					wCycleCount := wCycleCount + 1;
					IF (wCycleCount > wMotorTimeOn) OR GVL_IO.CircMotorLimit[FTN10,GVL.iPlus] OR
							GVL_IO.CircMotorLimit[FTN10,GVL.iMinus] THEN	//done with timer or any limit activated
						GVL_IO.CircMotorRelay[FTN10,GVL.iPlus] := FALSE;		//turn off outputs
						GVL_IO.CircMotorRelay[FTN10,GVL.iMinus] := FALSE;
						GVL.mb_Output_Coils[GVL.REALTIME_ADVANCE] := FALSE; // reset the advance boolean
						wCycleCount := 0;					//reset the timer counter						
						nRawFBpos	:=	GVL_IO.CircMotorPot[FTN10];
						nActualPos		:= 	LREAL_TO_DINT(
							INT_TO_LREAL(GVL.w_RegisterConfig[Index,GVL.iCIRC,0 ]) +						//base is min position
							(((INT_TO_LREAL(nRawFBpos - GVL.w_RegisterConfig[Index,GVL.iCIRC,2 ])) 			//voltage offset from low calibration
							* 	(INT_TO_LREAL(GVL.w_RegisterConfig[Index,GVL.iCIRC,1 ] - GVL.w_RegisterConfig[Index,GVL.iCIRC,0 ])))	//total position length
							/	( INT_TO_LREAL(GVL.w_RegisterConfig[Index,GVL.iCIRC,3 ] - GVL.w_RegisterConfig[Index,GVL.iCIRC,2 ])))	//total voltage range
							);
						GVL.mb_Output_Registers[w_temp_index+(GVL.iActualPosition)]	:= 
								DINT_TO_WORD(nActualPos);		//post the scaled actual position here to OUTPUT

					END_IF
				END_IF
			END_IF
			IF GVL.mb_Output_Coils[GVL.REALTIME_RETARD] THEN
				IF GVL_IO.CircMotorPot[FTN10] > 800 THEN				//test the FB for limit - assumes 32767 is max of 10 VDC
					GVL_IO.CircMotorRelay[FTN10,GVL.iPlus] := FALSE;				// turn on the reverse output
					GVL_IO.CircMotorRelay[FTN10,GVL.iMinus] := TRUE;
					wCycleCount := wCycleCount + 1;
					IF (wCycleCount > wMotorTimeOn) OR GVL_IO.CircMotorLimit[FTN10,GVL.iPlus] OR
							GVL_IO.CircMotorLimit[FTN10,GVL.iMinus] THEN	//done with timer or any limit activated
						GVL_IO.CircMotorRelay[FTN10,GVL.iPlus] := FALSE;		//turn off outputs
						GVL_IO.CircMotorRelay[FTN10,GVL.iMinus] := FALSE;
						GVL.mb_Output_Coils[GVL.REALTIME_RETARD] := FALSE; // reset the reverse boolean
						wCycleCount := 0;					//reset the timer counter						
						nRawFBpos	:=	GVL_IO.CircMotorPot[FTN10];
						nActualPos		:= 	LREAL_TO_DINT(
							INT_TO_LREAL(GVL.w_RegisterConfig[Index,GVL.iCIRC,0 ]) +						//base is min position
							(((INT_TO_LREAL(nRawFBpos - GVL.w_RegisterConfig[Index,GVL.iCIRC,2 ])) 			//voltage offset from low calibration
							* 	(INT_TO_LREAL(GVL.w_RegisterConfig[Index,GVL.iCIRC,1 ] - GVL.w_RegisterConfig[Index,GVL.iCIRC,0 ])))	//total position length
							/	( INT_TO_LREAL(GVL.w_RegisterConfig[Index,GVL.iCIRC,3 ] - GVL.w_RegisterConfig[Index,GVL.iCIRC,2 ])))	//total voltage range
							);
						GVL.mb_Output_Registers[w_temp_index+(GVL.iActualPosition)]	:= 
								DINT_TO_WORD(nActualPos);		//post the scaled actual position here to OUTPUT
					END_IF
				END_IF
			END_IF
	 32:	//Lateral FB Ftn 1
			GVL.mb_Output_Registers[GVL.REALTIME_PLC_A2D] :=	INT_TO_WORD(GVL_IO.LateralMotorPot[FTN1]);
			w_temp_index	:= GVL.RUNREG_START+(GVL.RUNREG_SIZE*3*FTN1)+(GVL.RUNREG_SIZE*GVL.iLAT);
			IF GVL.mb_Output_Coils[GVL.REALTIME_ADVANCE] THEN		//move the motor forward
				IF GVL_IO.LateralMotorPot[FTN1] < 32000 THEN				//test the FB for limit - assumes 32767 is max of 10 VDC
					GVL_IO.LateralMotorRelay[FTN1,GVL.iPlus] := TRUE;				// turn on the advance output
					GVL_IO.LateralMotorRelay[FTN1,GVL.iMinus] := FALSE;
					wCycleCount := wCycleCount + 1;
					IF (wCycleCount > wMotorTimeOn) OR GVL_IO.LateralMotorLimit[FTN1,GVL.iPlus] OR
							GVL_IO.LateralMotorLimit[FTN1,GVL.iMinus] THEN	//done with timer or any limit activated
						GVL_IO.LateralMotorRelay[FTN1,GVL.iPlus] := FALSE;		//turn off outputs
						GVL_IO.LateralMotorRelay[FTN1,GVL.iMinus] := FALSE;
						GVL.mb_Output_Coils[GVL.REALTIME_ADVANCE] := FALSE; // reset the advance boolean
						wCycleCount := 0;					//reset the timer counter						
						nRawFBpos	:=	GVL_IO.LateralMotorPot[FTN1];
						nActualPos		:= 	LREAL_TO_DINT(
							INT_TO_LREAL(GVL.w_RegisterConfig[Index,GVL.iLAT,0 ]) +							//base is min position
							(((INT_TO_LREAL(nRawFBpos - GVL.w_RegisterConfig[Index,GVL.iLAT,2 ])) 			//voltage offset from low calibration
							* 	(INT_TO_LREAL(GVL.w_RegisterConfig[Index,GVL.iLAT,1 ] - GVL.w_RegisterConfig[Index,GVL.iLAT,0 ])))	//total position length
							/	( INT_TO_LREAL(GVL.w_RegisterConfig[Index,GVL.iLAT,3 ] - GVL.w_RegisterConfig[Index,GVL.iLAT,2 ])))	//total voltage range
							);
						GVL.mb_Output_Registers[w_temp_index+(GVL.iActualPosition)]	:= 
								DINT_TO_WORD(nActualPos);		//post the scaled actual position here to OUTPUT

					END_IF
				END_IF
			END_IF
			IF GVL.mb_Output_Coils[GVL.REALTIME_RETARD] THEN
				IF GVL_IO.LateralMotorPot[FTN1] > 800 THEN				//test the FB for limit - assumes 32767 is max of 10 VDC
					GVL_IO.LateralMotorRelay[FTN1,GVL.iPlus] := FALSE;				// turn on the reverse output
					GVL_IO.LateralMotorRelay[FTN1,GVL.iMinus] := TRUE;
					wCycleCount := wCycleCount + 1;
					IF (wCycleCount > wMotorTimeOn) OR GVL_IO.LateralMotorLimit[FTN1,GVL.iPlus] OR
							GVL_IO.LateralMotorLimit[FTN1,GVL.iMinus] THEN	//done with timer or any limit activated
						GVL_IO.LateralMotorRelay[FTN1,GVL.iPlus] := FALSE;		//turn off outputs
						GVL_IO.LateralMotorRelay[FTN1,GVL.iMinus] := FALSE;
						GVL.mb_Output_Coils[GVL.REALTIME_RETARD] := FALSE; // reset the reverse boolean
						wCycleCount := 0;					//reset the timer counter						
						nRawFBpos	:=	GVL_IO.LateralMotorPot[FTN1];
						nActualPos		:= 	LREAL_TO_DINT(
							INT_TO_LREAL(GVL.w_RegisterConfig[Index,GVL.iLAT,0 ]) +							//base is min position
							(((INT_TO_LREAL(nRawFBpos - GVL.w_RegisterConfig[Index,GVL.iLAT,2 ])) 			//voltage offset from low calibration
							* 	(INT_TO_LREAL(GVL.w_RegisterConfig[Index,GVL.iLAT,1 ] - GVL.w_RegisterConfig[Index,GVL.iLAT,0 ])))	//total position length
							/	( INT_TO_LREAL(GVL.w_RegisterConfig[Index,GVL.iLAT,3 ] - GVL.w_RegisterConfig[Index,GVL.iLAT,2 ])))	//total voltage range
							);
						GVL.mb_Output_Registers[w_temp_index+(GVL.iActualPosition)]	:= 
								DINT_TO_WORD(nActualPos);		//post the scaled actual position here to OUTPUT
					END_IF
				END_IF
			END_IF
	 33:	//Lateral FB Ftn 2
			GVL.mb_Output_Registers[GVL.REALTIME_PLC_A2D] :=	INT_TO_WORD(GVL_IO.LateralMotorPot[FTN2]);
			w_temp_index	:= GVL.RUNREG_START+(GVL.RUNREG_SIZE*3*FTN2)+(GVL.RUNREG_SIZE*GVL.iLAT);
			IF GVL.mb_Output_Coils[GVL.REALTIME_ADVANCE] THEN		//move the motor forward
				IF GVL_IO.LateralMotorPot[FTN2] < 32000 THEN				//test the FB for limit - assumes 32767 is max of 10 VDC
					GVL_IO.LateralMotorRelay[FTN2,GVL.iPlus] := TRUE;				// turn on the advance output
					GVL_IO.LateralMotorRelay[FTN2,GVL.iMinus] := FALSE;
					wCycleCount := wCycleCount + 1;
					IF (wCycleCount > wMotorTimeOn) OR GVL_IO.LateralMotorLimit[FTN2,GVL.iPlus] OR
							GVL_IO.LateralMotorLimit[FTN2,GVL.iMinus] THEN	//done with timer or any limit activated
						GVL_IO.LateralMotorRelay[FTN2,GVL.iPlus] := FALSE;		//turn off outputs
						GVL_IO.LateralMotorRelay[FTN2,GVL.iMinus] := FALSE;
						GVL.mb_Output_Coils[GVL.REALTIME_ADVANCE] := FALSE; // reset the advance boolean
						wCycleCount := 0;					//reset the timer counter						
						nRawFBpos	:=	GVL_IO.LateralMotorPot[FTN2];
						nActualPos		:= 	LREAL_TO_DINT(
							INT_TO_LREAL(GVL.w_RegisterConfig[Index,GVL.iLAT,0 ]) +							//base is min position
							(((INT_TO_LREAL(nRawFBpos - GVL.w_RegisterConfig[Index,GVL.iLAT,2 ])) 			//voltage offset from low calibration
							* 	(INT_TO_LREAL(GVL.w_RegisterConfig[Index,GVL.iLAT,1 ] - GVL.w_RegisterConfig[Index,GVL.iLAT,0 ])))	//total position length
							/	( INT_TO_LREAL(GVL.w_RegisterConfig[Index,GVL.iLAT,3 ] - GVL.w_RegisterConfig[Index,GVL.iLAT,2 ])))	//total voltage range
							);
						GVL.mb_Output_Registers[w_temp_index+(GVL.iActualPosition)]	:= 
								DINT_TO_WORD(nActualPos);		//post the scaled actual position here to OUTPUT

					END_IF
				END_IF
			END_IF
			IF GVL.mb_Output_Coils[GVL.REALTIME_RETARD] THEN
				IF GVL_IO.LateralMotorPot[FTN2] > 800 THEN				//test the FB for limit - assumes 32767 is max of 10 VDC
					GVL_IO.LateralMotorRelay[FTN2,GVL.iPlus] := FALSE;				// turn on the reverse output
					GVL_IO.LateralMotorRelay[FTN2,GVL.iMinus] := TRUE;
					wCycleCount := wCycleCount + 1;
					IF (wCycleCount > wMotorTimeOn) OR GVL_IO.LateralMotorLimit[FTN2,GVL.iPlus] OR
							GVL_IO.LateralMotorLimit[FTN2,GVL.iMinus] THEN	//done with timer or any limit activated
						GVL_IO.LateralMotorRelay[FTN2,GVL.iPlus] := FALSE;		//turn off outputs
						GVL_IO.LateralMotorRelay[FTN2,GVL.iMinus] := FALSE;
						GVL.mb_Output_Coils[GVL.REALTIME_RETARD] := FALSE; // reset the reverse boolean
						wCycleCount := 0;					//reset the timer counter						
						nRawFBpos	:=	GVL_IO.LateralMotorPot[FTN2];
						nActualPos		:= 	LREAL_TO_DINT(
							INT_TO_LREAL(GVL.w_RegisterConfig[Index,GVL.iLAT,0 ]) +							//base is min position
							(((INT_TO_LREAL(nRawFBpos - GVL.w_RegisterConfig[Index,GVL.iLAT,2 ])) 			//voltage offset from low calibration
							* 	(INT_TO_LREAL(GVL.w_RegisterConfig[Index,GVL.iLAT,1 ] - GVL.w_RegisterConfig[Index,GVL.iLAT,0 ])))	//total position length
							/	( INT_TO_LREAL(GVL.w_RegisterConfig[Index,GVL.iLAT,3 ] - GVL.w_RegisterConfig[Index,GVL.iLAT,2 ])))	//total voltage range
							);
						GVL.mb_Output_Registers[w_temp_index+(GVL.iActualPosition)]	:= 
								DINT_TO_WORD(nActualPos);		//post the scaled actual position here to OUTPUT
					END_IF
				END_IF
			END_IF
	 34:	//Lateral FB Ftn 3
			GVL.mb_Output_Registers[GVL.REALTIME_PLC_A2D] :=	INT_TO_WORD(GVL_IO.LateralMotorPot[FTN3]);
			w_temp_index	:= GVL.RUNREG_START+(GVL.RUNREG_SIZE*3*FTN3)+(GVL.RUNREG_SIZE*GVL.iLAT);
			IF GVL.mb_Output_Coils[GVL.REALTIME_ADVANCE] THEN		//move the motor forward
				IF GVL_IO.LateralMotorPot[FTN3] < 32000 THEN				//test the FB for limit - assumes 32767 is max of 10 VDC
					GVL_IO.LateralMotorRelay[FTN3,GVL.iPlus] := TRUE;				// turn on the advance output
					GVL_IO.LateralMotorRelay[FTN3,GVL.iMinus] := FALSE;
					wCycleCount := wCycleCount + 1;
					IF (wCycleCount > wMotorTimeOn) OR GVL_IO.LateralMotorLimit[FTN3,GVL.iPlus] OR
							GVL_IO.LateralMotorLimit[FTN3,GVL.iMinus] THEN	//done with timer or any limit activated
						GVL_IO.LateralMotorRelay[FTN3,GVL.iPlus] := FALSE;		//turn off outputs
						GVL_IO.LateralMotorRelay[FTN3,GVL.iMinus] := FALSE;
						GVL.mb_Output_Coils[GVL.REALTIME_ADVANCE] := FALSE; // reset the advance boolean
						wCycleCount := 0;					//reset the timer counter						
						nRawFBpos	:=	GVL_IO.LateralMotorPot[FTN3];
						nActualPos		:= 	LREAL_TO_DINT(
							INT_TO_LREAL(GVL.w_RegisterConfig[Index,GVL.iLAT,0 ]) +							//base is min position
							(((INT_TO_LREAL(nRawFBpos - GVL.w_RegisterConfig[Index,GVL.iLAT,2 ])) 			//voltage offset from low calibration
							* 	(INT_TO_LREAL(GVL.w_RegisterConfig[Index,GVL.iLAT,1 ] - GVL.w_RegisterConfig[Index,GVL.iLAT,0 ])))	//total position length
							/	( INT_TO_LREAL(GVL.w_RegisterConfig[Index,GVL.iLAT,3 ] - GVL.w_RegisterConfig[Index,GVL.iLAT,2 ])))	//total voltage range
							);
						GVL.mb_Output_Registers[w_temp_index+(GVL.iActualPosition)]	:= 
								DINT_TO_WORD(nActualPos);		//post the scaled actual position here to OUTPUT

					END_IF
				END_IF
			END_IF
			IF GVL.mb_Output_Coils[GVL.REALTIME_RETARD] THEN
				IF GVL_IO.LateralMotorPot[FTN3] > 800 THEN				//test the FB for limit - assumes 32767 is max of 10 VDC
					GVL_IO.LateralMotorRelay[FTN3,GVL.iPlus] := FALSE;				// turn on the reverse output
					GVL_IO.LateralMotorRelay[FTN3,GVL.iMinus] := TRUE;
					wCycleCount := wCycleCount + 1;
					IF (wCycleCount > wMotorTimeOn) OR GVL_IO.LateralMotorLimit[FTN3,GVL.iPlus] OR
							GVL_IO.LateralMotorLimit[FTN3,GVL.iMinus] THEN	//done with timer or any limit activated
						GVL_IO.LateralMotorRelay[FTN3,GVL.iPlus] := FALSE;		//turn off outputs
						GVL_IO.LateralMotorRelay[FTN3,GVL.iMinus] := FALSE;
						GVL.mb_Output_Coils[GVL.REALTIME_RETARD] := FALSE; // reset the reverse boolean
						wCycleCount := 0;					//reset the timer counter						
						nRawFBpos	:=	GVL_IO.LateralMotorPot[FTN3];
						nActualPos		:= 	LREAL_TO_DINT(
							INT_TO_LREAL(GVL.w_RegisterConfig[Index,GVL.iLAT,0 ]) +							//base is min position
							(((INT_TO_LREAL(nRawFBpos - GVL.w_RegisterConfig[Index,GVL.iLAT,2 ])) 			//voltage offset from low calibration
							* 	(INT_TO_LREAL(GVL.w_RegisterConfig[Index,GVL.iLAT,1 ] - GVL.w_RegisterConfig[Index,GVL.iLAT,0 ])))	//total position length
							/	( INT_TO_LREAL(GVL.w_RegisterConfig[Index,GVL.iLAT,3 ] - GVL.w_RegisterConfig[Index,GVL.iLAT,2 ])))	//total voltage range
							);
						GVL.mb_Output_Registers[w_temp_index+(GVL.iActualPosition)]	:= 
								DINT_TO_WORD(nActualPos);		//post the scaled actual position here to OUTPUT
					END_IF
				END_IF
			END_IF
	 35:	//Lateral FB Ftn 4
			GVL.mb_Output_Registers[GVL.REALTIME_PLC_A2D] :=	INT_TO_WORD(GVL_IO.LateralMotorPot[FTN4]);
			w_temp_index	:= GVL.RUNREG_START+(GVL.RUNREG_SIZE*3*FTN4)+(GVL.RUNREG_SIZE*GVL.iLAT);
			IF GVL.mb_Output_Coils[GVL.REALTIME_ADVANCE] THEN		//move the motor forward
				IF GVL_IO.LateralMotorPot[FTN4] < 32000 THEN				//test the FB for limit - assumes 32767 is max of 10 VDC
					GVL_IO.LateralMotorRelay[FTN4,GVL.iPlus] := TRUE;				// turn on the advance output
					GVL_IO.LateralMotorRelay[FTN4,GVL.iMinus] := FALSE;
					wCycleCount := wCycleCount + 1;
					IF (wCycleCount > wMotorTimeOn) OR GVL_IO.LateralMotorLimit[FTN4,GVL.iPlus] OR
							GVL_IO.LateralMotorLimit[FTN4,GVL.iMinus] THEN	//done with timer or any limit activated
						GVL_IO.LateralMotorRelay[FTN4,GVL.iPlus] := FALSE;		//turn off outputs
						GVL_IO.LateralMotorRelay[FTN4,GVL.iMinus] := FALSE;
						GVL.mb_Output_Coils[GVL.REALTIME_ADVANCE] := FALSE; // reset the advance boolean
						wCycleCount := 0;					//reset the timer counter						
						nRawFBpos	:=	GVL_IO.LateralMotorPot[FTN4];
						nActualPos		:= 	LREAL_TO_DINT(
							INT_TO_LREAL(GVL.w_RegisterConfig[Index,GVL.iLAT,0 ]) +							//base is min position
							(((INT_TO_LREAL(nRawFBpos - GVL.w_RegisterConfig[Index,GVL.iLAT,2 ])) 			//voltage offset from low calibration
							* 	(INT_TO_LREAL(GVL.w_RegisterConfig[Index,GVL.iLAT,1 ] - GVL.w_RegisterConfig[Index,GVL.iLAT,0 ])))	//total position length
							/	( INT_TO_LREAL(GVL.w_RegisterConfig[Index,GVL.iLAT,3 ] - GVL.w_RegisterConfig[Index,GVL.iLAT,2 ])))	//total voltage range
							);
						GVL.mb_Output_Registers[w_temp_index+(GVL.iActualPosition)]	:= 
								DINT_TO_WORD(nActualPos);		//post the scaled actual position here to OUTPUT

					END_IF
				END_IF
			END_IF
			IF GVL.mb_Output_Coils[GVL.REALTIME_RETARD] THEN
				IF GVL_IO.LateralMotorPot[FTN4] > 800 THEN				//test the FB for limit - assumes 32767 is max of 10 VDC
					GVL_IO.LateralMotorRelay[FTN4,GVL.iPlus] := FALSE;				// turn on the reverse output
					GVL_IO.LateralMotorRelay[FTN4,GVL.iMinus] := TRUE;
					wCycleCount := wCycleCount + 1;
					IF (wCycleCount > wMotorTimeOn) OR GVL_IO.LateralMotorLimit[FTN4,GVL.iPlus] OR
							GVL_IO.LateralMotorLimit[FTN4,GVL.iMinus] THEN	//done with timer or any limit activated
						GVL_IO.LateralMotorRelay[FTN4,GVL.iPlus] := FALSE;		//turn off outputs
						GVL_IO.LateralMotorRelay[FTN4,GVL.iMinus] := FALSE;
						GVL.mb_Output_Coils[GVL.REALTIME_RETARD] := FALSE; // reset the reverse boolean
						wCycleCount := 0;					//reset the timer counter						
						nRawFBpos	:=	GVL_IO.LateralMotorPot[FTN4];
						nActualPos		:= 	LREAL_TO_DINT(
							INT_TO_LREAL(GVL.w_RegisterConfig[Index,GVL.iLAT,0 ]) +							//base is min position
							(((INT_TO_LREAL(nRawFBpos - GVL.w_RegisterConfig[Index,GVL.iLAT,2 ])) 			//voltage offset from low calibration
							* 	(INT_TO_LREAL(GVL.w_RegisterConfig[Index,GVL.iLAT,1 ] - GVL.w_RegisterConfig[Index,GVL.iLAT,0 ])))	//total position length
							/	( INT_TO_LREAL(GVL.w_RegisterConfig[Index,GVL.iLAT,3 ] - GVL.w_RegisterConfig[Index,GVL.iLAT,2 ])))	//total voltage range
							);
						GVL.mb_Output_Registers[w_temp_index+(GVL.iActualPosition)]	:= 
								DINT_TO_WORD(nActualPos);		//post the scaled actual position here to OUTPUT
					END_IF
				END_IF
			END_IF
	 36:	//Lateral FB Ftn 5
			GVL.mb_Output_Registers[GVL.REALTIME_PLC_A2D] :=	INT_TO_WORD(GVL_IO.LateralMotorPot[FTN5]);
			w_temp_index	:= GVL.RUNREG_START+(GVL.RUNREG_SIZE*3*FTN5)+(GVL.RUNREG_SIZE*GVL.iLAT);
			IF GVL.mb_Output_Coils[GVL.REALTIME_ADVANCE] THEN		//move the motor forward
				IF GVL_IO.LateralMotorPot[FTN5] < 32000 THEN				//test the FB for limit - assumes 32767 is max of 10 VDC
					GVL_IO.LateralMotorRelay[FTN5,GVL.iPlus] := TRUE;				// turn on the advance output
					GVL_IO.LateralMotorRelay[FTN5,GVL.iMinus] := FALSE;
					wCycleCount := wCycleCount + 1;
					IF (wCycleCount > wMotorTimeOn) OR GVL_IO.LateralMotorLimit[FTN5,GVL.iPlus] OR
							GVL_IO.LateralMotorLimit[FTN5,GVL.iMinus] THEN	//done with timer or any limit activated
						GVL_IO.LateralMotorRelay[FTN5,GVL.iPlus] := FALSE;		//turn off outputs
						GVL_IO.LateralMotorRelay[FTN5,GVL.iMinus] := FALSE;
						GVL.mb_Output_Coils[GVL.REALTIME_ADVANCE] := FALSE; // reset the advance boolean
						wCycleCount := 0;					//reset the timer counter						
						nRawFBpos	:=	GVL_IO.LateralMotorPot[FTN5];
						nActualPos		:= 	LREAL_TO_DINT(
							INT_TO_LREAL(GVL.w_RegisterConfig[Index,GVL.iLAT,0 ]) +							//base is min position
							(((INT_TO_LREAL(nRawFBpos - GVL.w_RegisterConfig[Index,GVL.iLAT,2 ])) 			//voltage offset from low calibration
							* 	(INT_TO_LREAL(GVL.w_RegisterConfig[Index,GVL.iLAT,1 ] - GVL.w_RegisterConfig[Index,GVL.iLAT,0 ])))	//total position length
							/	( INT_TO_LREAL(GVL.w_RegisterConfig[Index,GVL.iLAT,3 ] - GVL.w_RegisterConfig[Index,GVL.iLAT,2 ])))	//total voltage range
							);
						GVL.mb_Output_Registers[w_temp_index+(GVL.iActualPosition)]	:= 
								DINT_TO_WORD(nActualPos);		//post the scaled actual position here to OUTPUT

					END_IF
				END_IF
			END_IF
			IF GVL.mb_Output_Coils[GVL.REALTIME_RETARD] THEN
				IF GVL_IO.LateralMotorPot[FTN5] > 800 THEN				//test the FB for limit - assumes 32767 is max of 10 VDC
					GVL_IO.LateralMotorRelay[FTN5,GVL.iPlus] := FALSE;				// turn on the reverse output
					GVL_IO.LateralMotorRelay[FTN5,GVL.iMinus] := TRUE;
					wCycleCount := wCycleCount + 1;
					IF (wCycleCount > wMotorTimeOn) OR GVL_IO.LateralMotorLimit[FTN5,GVL.iPlus] OR
							GVL_IO.LateralMotorLimit[FTN5,GVL.iMinus] THEN	//done with timer or any limit activated
						GVL_IO.LateralMotorRelay[FTN5,GVL.iPlus] := FALSE;		//turn off outputs
						GVL_IO.LateralMotorRelay[FTN5,GVL.iMinus] := FALSE;
						GVL.mb_Output_Coils[GVL.REALTIME_RETARD] := FALSE; // reset the reverse boolean
						wCycleCount := 0;					//reset the timer counter						
						nRawFBpos	:=	GVL_IO.LateralMotorPot[FTN5];
						nActualPos		:= 	LREAL_TO_DINT(
							INT_TO_LREAL(GVL.w_RegisterConfig[Index,GVL.iLAT,0 ]) +							//base is min position
							(((INT_TO_LREAL(nRawFBpos - GVL.w_RegisterConfig[Index,GVL.iLAT,2 ])) 			//voltage offset from low calibration
							* 	(INT_TO_LREAL(GVL.w_RegisterConfig[Index,GVL.iLAT,1 ] - GVL.w_RegisterConfig[Index,GVL.iLAT,0 ])))	//total position length
							/	( INT_TO_LREAL(GVL.w_RegisterConfig[Index,GVL.iLAT,3 ] - GVL.w_RegisterConfig[Index,GVL.iLAT,2 ])))	//total voltage range
							);
						GVL.mb_Output_Registers[w_temp_index+(GVL.iActualPosition)]	:= 
								DINT_TO_WORD(nActualPos);		//post the scaled actual position here to OUTPUT
					END_IF
				END_IF
			END_IF
	 37:	//Lateral FB Ftn 6
			GVL.mb_Output_Registers[GVL.REALTIME_PLC_A2D] :=	INT_TO_WORD(GVL_IO.LateralMotorPot[FTN6]);
		//	FTN 6 special
			w_temp_index	:= GVL.RUNREG_START+(GVL.RUNREG_SIZE*3*FTN6)+(GVL.RUNREG_SIZE*GVL.iLAT)+10;
			IF GVL.mb_Output_Coils[GVL.REALTIME_ADVANCE] THEN		//move the motor forward
				IF GVL_IO.LateralMotorPot[FTN6] < 32000 THEN				//test the FB for limit - assumes 32767 is max of 10 VDC
					GVL_IO.LateralMotorRelay[FTN6,GVL.iPlus] := TRUE;				// turn on the advance output
					GVL_IO.LateralMotorRelay[FTN6,GVL.iMinus] := FALSE;
					wCycleCount := wCycleCount + 1;
					IF (wCycleCount > wMotorTimeOn) OR GVL_IO.LateralMotorLimit[FTN6,GVL.iPlus] OR
							GVL_IO.LateralMotorLimit[FTN6,GVL.iMinus] THEN	//done with timer or any limit activated
						GVL_IO.LateralMotorRelay[FTN6,GVL.iPlus] := FALSE;		//turn off outputs
						GVL_IO.LateralMotorRelay[FTN6,GVL.iMinus] := FALSE;
						GVL.mb_Output_Coils[GVL.REALTIME_ADVANCE] := FALSE; // reset the advance boolean
						wCycleCount := 0;					//reset the timer counter						
						nRawFBpos	:=	GVL_IO.LateralMotorPot[FTN6];
						nActualPos		:= 	LREAL_TO_DINT(
							INT_TO_LREAL(GVL.w_RegisterConfig[Index,GVL.iLAT,0 ]) +							//base is min position
							(((INT_TO_LREAL(nRawFBpos - GVL.w_RegisterConfig[Index,GVL.iLAT,2 ])) 			//voltage offset from low calibration
							* 	(INT_TO_LREAL(GVL.w_RegisterConfig[Index,GVL.iLAT,1 ] - GVL.w_RegisterConfig[Index,GVL.iLAT,0 ])))	//total position length
							/	( INT_TO_LREAL(GVL.w_RegisterConfig[Index,GVL.iLAT,3 ] - GVL.w_RegisterConfig[Index,GVL.iLAT,2 ])))	//total voltage range
							);
						GVL.mb_Output_Registers[w_temp_index+(GVL.iActualPosition)]	:= 
								DINT_TO_WORD(nActualPos);		//post the scaled actual position here to OUTPUT

